   // UNICODE_TO_GBK[9822] := 16#5E62;
   // UNICODE_TO_GBK[9823] := 16#B4B1;
   // UNICODE_TO_GBK[9824] := 16#5E63;
   // UNICODE_TO_GBK[9825] := 16#8EC5;
   // UNICODE_TO_GBK[9826] := 16#5E64;
   // UNICODE_TO_GBK[9827] := 16#8EC6;
   // UNICODE_TO_GBK[9828] := 16#5E65;
   // UNICODE_TO_GBK[9829] := 16#8EC7;
   // UNICODE_TO_GBK[9830] := 16#5E66;
   // UNICODE_TO_GBK[9831] := 16#8EC8;
   // UNICODE_TO_GBK[9832] := 16#5E67;
   // UNICODE_TO_GBK[9833] := 16#8EC9;
   // UNICODE_TO_GBK[9834] := 16#5E68;
   // UNICODE_TO_GBK[9835] := 16#8ECA;
   // UNICODE_TO_GBK[9836] := 16#5E69;
   // UNICODE_TO_GBK[9837] := 16#8ECB;
   // UNICODE_TO_GBK[9838] := 16#5E6A;
   // UNICODE_TO_GBK[9839] := 16#8ECC;
   // UNICODE_TO_GBK[9840] := 16#5E6B;
   // UNICODE_TO_GBK[9841] := 16#8ECD;
   // UNICODE_TO_GBK[9842] := 16#5E6C;
   // UNICODE_TO_GBK[9843] := 16#8ECE;
   // UNICODE_TO_GBK[9844] := 16#5E6D;
   // UNICODE_TO_GBK[9845] := 16#8ECF;
   // UNICODE_TO_GBK[9846] := 16#5E6E;
   // UNICODE_TO_GBK[9847] := 16#8ED0;
   // UNICODE_TO_GBK[9848] := 16#5E6F;
   // UNICODE_TO_GBK[9849] := 16#8ED1;
   // UNICODE_TO_GBK[9850] := 16#5E70;
   // UNICODE_TO_GBK[9851] := 16#8ED2;
   // UNICODE_TO_GBK[9852] := 16#5E71;
   // UNICODE_TO_GBK[9853] := 16#8ED3;
   // UNICODE_TO_GBK[9854] := 16#5E72;
   // UNICODE_TO_GBK[9855] := 16#B8C9;
   // UNICODE_TO_GBK[9856] := 16#5E73;
   // UNICODE_TO_GBK[9857] := 16#C6BD;
   // UNICODE_TO_GBK[9858] := 16#5E74;
   // UNICODE_TO_GBK[9859] := 16#C4EA;
   // UNICODE_TO_GBK[9860] := 16#5E75;
   // UNICODE_TO_GBK[9861] := 16#8ED4;
   // UNICODE_TO_GBK[9862] := 16#5E76;
   // UNICODE_TO_GBK[9863] := 16#B2A2;
   // UNICODE_TO_GBK[9864] := 16#5E77;
   // UNICODE_TO_GBK[9865] := 16#8ED5;
   // UNICODE_TO_GBK[9866] := 16#5E78;
   // UNICODE_TO_GBK[9867] := 16#D0D2;
   // UNICODE_TO_GBK[9868] := 16#5E79;
   // UNICODE_TO_GBK[9869] := 16#8ED6;
   // UNICODE_TO_GBK[9870] := 16#5E7A;
   // UNICODE_TO_GBK[9871] := 16#E7DB;
   // UNICODE_TO_GBK[9872] := 16#5E7B;
   // UNICODE_TO_GBK[9873] := 16#BBC3;
   // UNICODE_TO_GBK[9874] := 16#5E7C;
   // UNICODE_TO_GBK[9875] := 16#D3D7;
   // UNICODE_TO_GBK[9876] := 16#5E7D;
   // UNICODE_TO_GBK[9877] := 16#D3C4;
   // UNICODE_TO_GBK[9878] := 16#5E7E;
   // UNICODE_TO_GBK[9879] := 16#8ED7;
   // UNICODE_TO_GBK[9880] := 16#5E7F;
   // UNICODE_TO_GBK[9881] := 16#B9E3;
   // UNICODE_TO_GBK[9882] := 16#5E80;
   // UNICODE_TO_GBK[9883] := 16#E2CF;
   // UNICODE_TO_GBK[9884] := 16#5E81;
   // UNICODE_TO_GBK[9885] := 16#8ED8;
   // UNICODE_TO_GBK[9886] := 16#5E82;
   // UNICODE_TO_GBK[9887] := 16#8ED9;
   // UNICODE_TO_GBK[9888] := 16#5E83;
   // UNICODE_TO_GBK[9889] := 16#8EDA;
   // UNICODE_TO_GBK[9890] := 16#5E84;
   // UNICODE_TO_GBK[9891] := 16#D7AF;
   // UNICODE_TO_GBK[9892] := 16#5E85;
   // UNICODE_TO_GBK[9893] := 16#8EDB;
   // UNICODE_TO_GBK[9894] := 16#5E86;
   // UNICODE_TO_GBK[9895] := 16#C7EC;
   // UNICODE_TO_GBK[9896] := 16#5E87;
   // UNICODE_TO_GBK[9897] := 16#B1D3;
   // UNICODE_TO_GBK[9898] := 16#5E88;
   // UNICODE_TO_GBK[9899] := 16#8EDC;
   // UNICODE_TO_GBK[9900] := 16#5E89;
   // UNICODE_TO_GBK[9901] := 16#8EDD;
   // UNICODE_TO_GBK[9902] := 16#5E8A;
   // UNICODE_TO_GBK[9903] := 16#B4B2;
   // UNICODE_TO_GBK[9904] := 16#5E8B;
   // UNICODE_TO_GBK[9905] := 16#E2D1;
   // UNICODE_TO_GBK[9906] := 16#5E8C;
   // UNICODE_TO_GBK[9907] := 16#8EDE;
   // UNICODE_TO_GBK[9908] := 16#5E8D;
   // UNICODE_TO_GBK[9909] := 16#8EDF;
   // UNICODE_TO_GBK[9910] := 16#5E8E;
   // UNICODE_TO_GBK[9911] := 16#8EE0;
   // UNICODE_TO_GBK[9912] := 16#5E8F;
   // UNICODE_TO_GBK[9913] := 16#D0F2;
   // UNICODE_TO_GBK[9914] := 16#5E90;
   // UNICODE_TO_GBK[9915] := 16#C2AE;
   // UNICODE_TO_GBK[9916] := 16#5E91;
   // UNICODE_TO_GBK[9917] := 16#E2D0;
   // UNICODE_TO_GBK[9918] := 16#5E92;
   // UNICODE_TO_GBK[9919] := 16#8EE1;
   // UNICODE_TO_GBK[9920] := 16#5E93;
   // UNICODE_TO_GBK[9921] := 16#BFE2;
   // UNICODE_TO_GBK[9922] := 16#5E94;
   // UNICODE_TO_GBK[9923] := 16#D3A6;
   // UNICODE_TO_GBK[9924] := 16#5E95;
   // UNICODE_TO_GBK[9925] := 16#B5D7;
   // UNICODE_TO_GBK[9926] := 16#5E96;
   // UNICODE_TO_GBK[9927] := 16#E2D2;
   // UNICODE_TO_GBK[9928] := 16#5E97;
   // UNICODE_TO_GBK[9929] := 16#B5EA;
   // UNICODE_TO_GBK[9930] := 16#5E98;
   // UNICODE_TO_GBK[9931] := 16#8EE2;
   // UNICODE_TO_GBK[9932] := 16#5E99;
   // UNICODE_TO_GBK[9933] := 16#C3ED;
   // UNICODE_TO_GBK[9934] := 16#5E9A;
   // UNICODE_TO_GBK[9935] := 16#B8FD;
   // UNICODE_TO_GBK[9936] := 16#5E9B;
   // UNICODE_TO_GBK[9937] := 16#8EE3;
   // UNICODE_TO_GBK[9938] := 16#5E9C;
   // UNICODE_TO_GBK[9939] := 16#B8AE;
   // UNICODE_TO_GBK[9940] := 16#5E9D;
   // UNICODE_TO_GBK[9941] := 16#8EE4;
   // UNICODE_TO_GBK[9942] := 16#5E9E;
   // UNICODE_TO_GBK[9943] := 16#C5D3;
   // UNICODE_TO_GBK[9944] := 16#5E9F;
   // UNICODE_TO_GBK[9945] := 16#B7CF;
   // UNICODE_TO_GBK[9946] := 16#5EA0;
   // UNICODE_TO_GBK[9947] := 16#E2D4;
   // UNICODE_TO_GBK[9948] := 16#5EA1;
   // UNICODE_TO_GBK[9949] := 16#8EE5;
   // UNICODE_TO_GBK[9950] := 16#5EA2;
   // UNICODE_TO_GBK[9951] := 16#8EE6;
   // UNICODE_TO_GBK[9952] := 16#5EA3;
   // UNICODE_TO_GBK[9953] := 16#8EE7;
   // UNICODE_TO_GBK[9954] := 16#5EA4;
   // UNICODE_TO_GBK[9955] := 16#8EE8;
   // UNICODE_TO_GBK[9956] := 16#5EA5;
   // UNICODE_TO_GBK[9957] := 16#E2D3;
   // UNICODE_TO_GBK[9958] := 16#5EA6;
   // UNICODE_TO_GBK[9959] := 16#B6C8;
   // UNICODE_TO_GBK[9960] := 16#5EA7;
   // UNICODE_TO_GBK[9961] := 16#D7F9;
   // UNICODE_TO_GBK[9962] := 16#5EA8;
   // UNICODE_TO_GBK[9963] := 16#8EE9;
   // UNICODE_TO_GBK[9964] := 16#5EA9;
   // UNICODE_TO_GBK[9965] := 16#8EEA;
   // UNICODE_TO_GBK[9966] := 16#5EAA;
   // UNICODE_TO_GBK[9967] := 16#8EEB;
   // UNICODE_TO_GBK[9968] := 16#5EAB;
   // UNICODE_TO_GBK[9969] := 16#8EEC;
   // UNICODE_TO_GBK[9970] := 16#5EAC;
   // UNICODE_TO_GBK[9971] := 16#8EED;
   // UNICODE_TO_GBK[9972] := 16#5EAD;
   // UNICODE_TO_GBK[9973] := 16#CDA5;
   // UNICODE_TO_GBK[9974] := 16#5EAE;
   // UNICODE_TO_GBK[9975] := 16#8EEE;
   // UNICODE_TO_GBK[9976] := 16#5EAF;
   // UNICODE_TO_GBK[9977] := 16#8EEF;
   // UNICODE_TO_GBK[9978] := 16#5EB0;
   // UNICODE_TO_GBK[9979] := 16#8EF0;
   // UNICODE_TO_GBK[9980] := 16#5EB1;
   // UNICODE_TO_GBK[9981] := 16#8EF1;
   // UNICODE_TO_GBK[9982] := 16#5EB2;
   // UNICODE_TO_GBK[9983] := 16#8EF2;
   // UNICODE_TO_GBK[9984] := 16#5EB3;
   // UNICODE_TO_GBK[9985] := 16#E2D8;
   // UNICODE_TO_GBK[9986] := 16#5EB4;
   // UNICODE_TO_GBK[9987] := 16#8EF3;
   // UNICODE_TO_GBK[9988] := 16#5EB5;
   // UNICODE_TO_GBK[9989] := 16#E2D6;
   // UNICODE_TO_GBK[9990] := 16#5EB6;
   // UNICODE_TO_GBK[9991] := 16#CAFC;
   // UNICODE_TO_GBK[9992] := 16#5EB7;
   // UNICODE_TO_GBK[9993] := 16#BFB5;
   // UNICODE_TO_GBK[9994] := 16#5EB8;
   // UNICODE_TO_GBK[9995] := 16#D3B9;
   // UNICODE_TO_GBK[9996] := 16#5EB9;
   // UNICODE_TO_GBK[9997] := 16#E2D5;
   // UNICODE_TO_GBK[9998] := 16#5EBA;
   // UNICODE_TO_GBK[9999] := 16#8EF4;
   // UNICODE_TO_GBK[10000] := 16#5EBB;
   // UNICODE_TO_GBK[10001] := 16#8EF5;
   // UNICODE_TO_GBK[10002] := 16#5EBC;
   // UNICODE_TO_GBK[10003] := 16#8EF6;
   // UNICODE_TO_GBK[10004] := 16#5EBD;
   // UNICODE_TO_GBK[10005] := 16#8EF7;
   // UNICODE_TO_GBK[10006] := 16#5EBE;
   // UNICODE_TO_GBK[10007] := 16#E2D7;
   // UNICODE_TO_GBK[10008] := 16#5EBF;
   // UNICODE_TO_GBK[10009] := 16#8EF8;
   // UNICODE_TO_GBK[10010] := 16#5EC0;
   // UNICODE_TO_GBK[10011] := 16#8EF9;
   // UNICODE_TO_GBK[10012] := 16#5EC1;
   // UNICODE_TO_GBK[10013] := 16#8EFA;
   // UNICODE_TO_GBK[10014] := 16#5EC2;
   // UNICODE_TO_GBK[10015] := 16#8EFB;
   // UNICODE_TO_GBK[10016] := 16#5EC3;
   // UNICODE_TO_GBK[10017] := 16#8EFC;
   // UNICODE_TO_GBK[10018] := 16#5EC4;
   // UNICODE_TO_GBK[10019] := 16#8EFD;
   // UNICODE_TO_GBK[10020] := 16#5EC5;
   // UNICODE_TO_GBK[10021] := 16#8EFE;
   // UNICODE_TO_GBK[10022] := 16#5EC6;
   // UNICODE_TO_GBK[10023] := 16#8F40;
   // UNICODE_TO_GBK[10024] := 16#5EC7;
   // UNICODE_TO_GBK[10025] := 16#8F41;
   // UNICODE_TO_GBK[10026] := 16#5EC8;
   // UNICODE_TO_GBK[10027] := 16#8F42;
   // UNICODE_TO_GBK[10028] := 16#5EC9;
   // UNICODE_TO_GBK[10029] := 16#C1AE;
   // UNICODE_TO_GBK[10030] := 16#5ECA;
   // UNICODE_TO_GBK[10031] := 16#C0C8;
   // UNICODE_TO_GBK[10032] := 16#5ECB;
   // UNICODE_TO_GBK[10033] := 16#8F43;
   // UNICODE_TO_GBK[10034] := 16#5ECC;
   // UNICODE_TO_GBK[10035] := 16#8F44;
   // UNICODE_TO_GBK[10036] := 16#5ECD;
   // UNICODE_TO_GBK[10037] := 16#8F45;
   // UNICODE_TO_GBK[10038] := 16#5ECE;
   // UNICODE_TO_GBK[10039] := 16#8F46;
   // UNICODE_TO_GBK[10040] := 16#5ECF;
   // UNICODE_TO_GBK[10041] := 16#8F47;
   // UNICODE_TO_GBK[10042] := 16#5ED0;
   // UNICODE_TO_GBK[10043] := 16#8F48;
   // UNICODE_TO_GBK[10044] := 16#5ED1;
   // UNICODE_TO_GBK[10045] := 16#E2DB;
   // UNICODE_TO_GBK[10046] := 16#5ED2;
   // UNICODE_TO_GBK[10047] := 16#E2DA;
   // UNICODE_TO_GBK[10048] := 16#5ED3;
   // UNICODE_TO_GBK[10049] := 16#C0AA;
   // UNICODE_TO_GBK[10050] := 16#5ED4;
   // UNICODE_TO_GBK[10051] := 16#8F49;
   // UNICODE_TO_GBK[10052] := 16#5ED5;
   // UNICODE_TO_GBK[10053] := 16#8F4A;
   // UNICODE_TO_GBK[10054] := 16#5ED6;
   // UNICODE_TO_GBK[10055] := 16#C1CE;
   // UNICODE_TO_GBK[10056] := 16#5ED7;
   // UNICODE_TO_GBK[10057] := 16#8F4B;
   // UNICODE_TO_GBK[10058] := 16#5ED8;
   // UNICODE_TO_GBK[10059] := 16#8F4C;
   // UNICODE_TO_GBK[10060] := 16#5ED9;
   // UNICODE_TO_GBK[10061] := 16#8F4D;
   // UNICODE_TO_GBK[10062] := 16#5EDA;
   // UNICODE_TO_GBK[10063] := 16#8F4E;
   // UNICODE_TO_GBK[10064] := 16#5EDB;
   // UNICODE_TO_GBK[10065] := 16#E2DC;
   // UNICODE_TO_GBK[10066] := 16#5EDC;
   // UNICODE_TO_GBK[10067] := 16#8F4F;
   // UNICODE_TO_GBK[10068] := 16#5EDD;
   // UNICODE_TO_GBK[10069] := 16#8F50;
   // UNICODE_TO_GBK[10070] := 16#5EDE;
   // UNICODE_TO_GBK[10071] := 16#8F51;
   // UNICODE_TO_GBK[10072] := 16#5EDF;
   // UNICODE_TO_GBK[10073] := 16#8F52;
   // UNICODE_TO_GBK[10074] := 16#5EE0;
   // UNICODE_TO_GBK[10075] := 16#8F53;
   // UNICODE_TO_GBK[10076] := 16#5EE1;
   // UNICODE_TO_GBK[10077] := 16#8F54;
   // UNICODE_TO_GBK[10078] := 16#5EE2;
   // UNICODE_TO_GBK[10079] := 16#8F55;
   // UNICODE_TO_GBK[10080] := 16#5EE3;
   // UNICODE_TO_GBK[10081] := 16#8F56;
   // UNICODE_TO_GBK[10082] := 16#5EE4;
   // UNICODE_TO_GBK[10083] := 16#8F57;
   // UNICODE_TO_GBK[10084] := 16#5EE5;
   // UNICODE_TO_GBK[10085] := 16#8F58;
   // UNICODE_TO_GBK[10086] := 16#5EE6;
   // UNICODE_TO_GBK[10087] := 16#8F59;
   // UNICODE_TO_GBK[10088] := 16#5EE7;
   // UNICODE_TO_GBK[10089] := 16#8F5A;
   // UNICODE_TO_GBK[10090] := 16#5EE8;
   // UNICODE_TO_GBK[10091] := 16#E2DD;
   // UNICODE_TO_GBK[10092] := 16#5EE9;
   // UNICODE_TO_GBK[10093] := 16#8F5B;
   // UNICODE_TO_GBK[10094] := 16#5EEA;
   // UNICODE_TO_GBK[10095] := 16#E2DE;
   // UNICODE_TO_GBK[10096] := 16#5EEB;
   // UNICODE_TO_GBK[10097] := 16#8F5C;
   // UNICODE_TO_GBK[10098] := 16#5EEC;
   // UNICODE_TO_GBK[10099] := 16#8F5D;
   // UNICODE_TO_GBK[10100] := 16#5EED;
   // UNICODE_TO_GBK[10101] := 16#8F5E;
   // UNICODE_TO_GBK[10102] := 16#5EEE;
   // UNICODE_TO_GBK[10103] := 16#8F5F;
   // UNICODE_TO_GBK[10104] := 16#5EEF;
   // UNICODE_TO_GBK[10105] := 16#8F60;
   // UNICODE_TO_GBK[10106] := 16#5EF0;
   // UNICODE_TO_GBK[10107] := 16#8F61;
   // UNICODE_TO_GBK[10108] := 16#5EF1;
   // UNICODE_TO_GBK[10109] := 16#8F62;
   // UNICODE_TO_GBK[10110] := 16#5EF2;
   // UNICODE_TO_GBK[10111] := 16#8F63;
   // UNICODE_TO_GBK[10112] := 16#5EF3;
   // UNICODE_TO_GBK[10113] := 16#8F64;
   // UNICODE_TO_GBK[10114] := 16#5EF4;
   // UNICODE_TO_GBK[10115] := 16#DBC8;
   // UNICODE_TO_GBK[10116] := 16#5EF5;
   // UNICODE_TO_GBK[10117] := 16#8F65;
   // UNICODE_TO_GBK[10118] := 16#5EF6;
   // UNICODE_TO_GBK[10119] := 16#D1D3;
   // UNICODE_TO_GBK[10120] := 16#5EF7;
   // UNICODE_TO_GBK[10121] := 16#CDA2;
   // UNICODE_TO_GBK[10122] := 16#5EF8;
   // UNICODE_TO_GBK[10123] := 16#8F66;
   // UNICODE_TO_GBK[10124] := 16#5EF9;
   // UNICODE_TO_GBK[10125] := 16#8F67;
   // UNICODE_TO_GBK[10126] := 16#5EFA;
   // UNICODE_TO_GBK[10127] := 16#BDA8;
   // UNICODE_TO_GBK[10128] := 16#5EFB;
   // UNICODE_TO_GBK[10129] := 16#8F68;
   // UNICODE_TO_GBK[10130] := 16#5EFC;
   // UNICODE_TO_GBK[10131] := 16#8F69;
   // UNICODE_TO_GBK[10132] := 16#5EFD;
   // UNICODE_TO_GBK[10133] := 16#8F6A;
   // UNICODE_TO_GBK[10134] := 16#5EFE;
   // UNICODE_TO_GBK[10135] := 16#DEC3;
   // UNICODE_TO_GBK[10136] := 16#5EFF;
   // UNICODE_TO_GBK[10137] := 16#D8A5;
   // UNICODE_TO_GBK[10138] := 16#5F00;
   // UNICODE_TO_GBK[10139] := 16#BFAA;
   // UNICODE_TO_GBK[10140] := 16#5F01;
   // UNICODE_TO_GBK[10141] := 16#DBCD;
   // UNICODE_TO_GBK[10142] := 16#5F02;
   // UNICODE_TO_GBK[10143] := 16#D2EC;
   // UNICODE_TO_GBK[10144] := 16#5F03;
   // UNICODE_TO_GBK[10145] := 16#C6FA;
   // UNICODE_TO_GBK[10146] := 16#5F04;
   // UNICODE_TO_GBK[10147] := 16#C5AA;
   // UNICODE_TO_GBK[10148] := 16#5F05;
   // UNICODE_TO_GBK[10149] := 16#8F6B;
   // UNICODE_TO_GBK[10150] := 16#5F06;
   // UNICODE_TO_GBK[10151] := 16#8F6C;
   // UNICODE_TO_GBK[10152] := 16#5F07;
   // UNICODE_TO_GBK[10153] := 16#8F6D;
   // UNICODE_TO_GBK[10154] := 16#5F08;
   // UNICODE_TO_GBK[10155] := 16#DEC4;
   // UNICODE_TO_GBK[10156] := 16#5F09;
   // UNICODE_TO_GBK[10157] := 16#8F6E;
   // UNICODE_TO_GBK[10158] := 16#5F0A;
   // UNICODE_TO_GBK[10159] := 16#B1D7;
   // UNICODE_TO_GBK[10160] := 16#5F0B;
   // UNICODE_TO_GBK[10161] := 16#DFAE;
   // UNICODE_TO_GBK[10162] := 16#5F0C;
   // UNICODE_TO_GBK[10163] := 16#8F6F;
   // UNICODE_TO_GBK[10164] := 16#5F0D;
   // UNICODE_TO_GBK[10165] := 16#8F70;
   // UNICODE_TO_GBK[10166] := 16#5F0E;
   // UNICODE_TO_GBK[10167] := 16#8F71;
   // UNICODE_TO_GBK[10168] := 16#5F0F;
   // UNICODE_TO_GBK[10169] := 16#CABD;
   // UNICODE_TO_GBK[10170] := 16#5F10;
   // UNICODE_TO_GBK[10171] := 16#8F72;
   // UNICODE_TO_GBK[10172] := 16#5F11;
   // UNICODE_TO_GBK[10173] := 16#DFB1;
   // UNICODE_TO_GBK[10174] := 16#5F12;
   // UNICODE_TO_GBK[10175] := 16#8F73;
   // UNICODE_TO_GBK[10176] := 16#5F13;
   // UNICODE_TO_GBK[10177] := 16#B9AD;
   // UNICODE_TO_GBK[10178] := 16#5F14;
   // UNICODE_TO_GBK[10179] := 16#8F74;
   // UNICODE_TO_GBK[10180] := 16#5F15;
   // UNICODE_TO_GBK[10181] := 16#D2FD;
   // UNICODE_TO_GBK[10182] := 16#5F16;
   // UNICODE_TO_GBK[10183] := 16#8F75;
   // UNICODE_TO_GBK[10184] := 16#5F17;
   // UNICODE_TO_GBK[10185] := 16#B8A5;
   // UNICODE_TO_GBK[10186] := 16#5F18;
   // UNICODE_TO_GBK[10187] := 16#BAEB;
   // UNICODE_TO_GBK[10188] := 16#5F19;
   // UNICODE_TO_GBK[10189] := 16#8F76;
   // UNICODE_TO_GBK[10190] := 16#5F1A;
   // UNICODE_TO_GBK[10191] := 16#8F77;
   // UNICODE_TO_GBK[10192] := 16#5F1B;
   // UNICODE_TO_GBK[10193] := 16#B3DA;
   // UNICODE_TO_GBK[10194] := 16#5F1C;
   // UNICODE_TO_GBK[10195] := 16#8F78;
   // UNICODE_TO_GBK[10196] := 16#5F1D;
   // UNICODE_TO_GBK[10197] := 16#8F79;
   // UNICODE_TO_GBK[10198] := 16#5F1E;
   // UNICODE_TO_GBK[10199] := 16#8F7A;
   // UNICODE_TO_GBK[10200] := 16#5F1F;
   // UNICODE_TO_GBK[10201] := 16#B5DC;
   // UNICODE_TO_GBK[10202] := 16#5F20;
   // UNICODE_TO_GBK[10203] := 16#D5C5;
   // UNICODE_TO_GBK[10204] := 16#5F21;
   // UNICODE_TO_GBK[10205] := 16#8F7B;
   // UNICODE_TO_GBK[10206] := 16#5F22;
   // UNICODE_TO_GBK[10207] := 16#8F7C;
   // UNICODE_TO_GBK[10208] := 16#5F23;
   // UNICODE_TO_GBK[10209] := 16#8F7D;
   // UNICODE_TO_GBK[10210] := 16#5F24;
   // UNICODE_TO_GBK[10211] := 16#8F7E;
   // UNICODE_TO_GBK[10212] := 16#5F25;
   // UNICODE_TO_GBK[10213] := 16#C3D6;
   // UNICODE_TO_GBK[10214] := 16#5F26;
   // UNICODE_TO_GBK[10215] := 16#CFD2;
   // UNICODE_TO_GBK[10216] := 16#5F27;
   // UNICODE_TO_GBK[10217] := 16#BBA1;
   // UNICODE_TO_GBK[10218] := 16#5F28;
   // UNICODE_TO_GBK[10219] := 16#8F80;
   // UNICODE_TO_GBK[10220] := 16#5F29;
   // UNICODE_TO_GBK[10221] := 16#E5F3;
   // UNICODE_TO_GBK[10222] := 16#5F2A;
   // UNICODE_TO_GBK[10223] := 16#E5F2;
   // UNICODE_TO_GBK[10224] := 16#5F2B;
   // UNICODE_TO_GBK[10225] := 16#8F81;
   // UNICODE_TO_GBK[10226] := 16#5F2C;
   // UNICODE_TO_GBK[10227] := 16#8F82;
   // UNICODE_TO_GBK[10228] := 16#5F2D;
   // UNICODE_TO_GBK[10229] := 16#E5F4;
   // UNICODE_TO_GBK[10230] := 16#5F2E;
   // UNICODE_TO_GBK[10231] := 16#8F83;
   // UNICODE_TO_GBK[10232] := 16#5F2F;
   // UNICODE_TO_GBK[10233] := 16#CDE4;
   // UNICODE_TO_GBK[10234] := 16#5F30;
   // UNICODE_TO_GBK[10235] := 16#8F84;
   // UNICODE_TO_GBK[10236] := 16#5F31;
   // UNICODE_TO_GBK[10237] := 16#C8F5;
   // UNICODE_TO_GBK[10238] := 16#5F32;
   // UNICODE_TO_GBK[10239] := 16#8F85;
   // UNICODE_TO_GBK[10240] := 16#5F33;
   // UNICODE_TO_GBK[10241] := 16#8F86;
   // UNICODE_TO_GBK[10242] := 16#5F34;
   // UNICODE_TO_GBK[10243] := 16#8F87;
   // UNICODE_TO_GBK[10244] := 16#5F35;
   // UNICODE_TO_GBK[10245] := 16#8F88;
   // UNICODE_TO_GBK[10246] := 16#5F36;
   // UNICODE_TO_GBK[10247] := 16#8F89;
   // UNICODE_TO_GBK[10248] := 16#5F37;
   // UNICODE_TO_GBK[10249] := 16#8F8A;
   // UNICODE_TO_GBK[10250] := 16#5F38;
   // UNICODE_TO_GBK[10251] := 16#8F8B;
   // UNICODE_TO_GBK[10252] := 16#5F39;
   // UNICODE_TO_GBK[10253] := 16#B5AF;
   // UNICODE_TO_GBK[10254] := 16#5F3A;
   // UNICODE_TO_GBK[10255] := 16#C7BF;
   // UNICODE_TO_GBK[10256] := 16#5F3B;
   // UNICODE_TO_GBK[10257] := 16#8F8C;
   // UNICODE_TO_GBK[10258] := 16#5F3C;
   // UNICODE_TO_GBK[10259] := 16#E5F6;
   // UNICODE_TO_GBK[10260] := 16#5F3D;
   // UNICODE_TO_GBK[10261] := 16#8F8D;
   // UNICODE_TO_GBK[10262] := 16#5F3E;
   // UNICODE_TO_GBK[10263] := 16#8F8E;
   // UNICODE_TO_GBK[10264] := 16#5F3F;
   // UNICODE_TO_GBK[10265] := 16#8F8F;
   // UNICODE_TO_GBK[10266] := 16#5F40;
   // UNICODE_TO_GBK[10267] := 16#ECB0;
   // UNICODE_TO_GBK[10268] := 16#5F41;
   // UNICODE_TO_GBK[10269] := 16#8F90;
   // UNICODE_TO_GBK[10270] := 16#5F42;
   // UNICODE_TO_GBK[10271] := 16#8F91;
   // UNICODE_TO_GBK[10272] := 16#5F43;
   // UNICODE_TO_GBK[10273] := 16#8F92;
   // UNICODE_TO_GBK[10274] := 16#5F44;
   // UNICODE_TO_GBK[10275] := 16#8F93;
   // UNICODE_TO_GBK[10276] := 16#5F45;
   // UNICODE_TO_GBK[10277] := 16#8F94;
   // UNICODE_TO_GBK[10278] := 16#5F46;
   // UNICODE_TO_GBK[10279] := 16#8F95;
   // UNICODE_TO_GBK[10280] := 16#5F47;
   // UNICODE_TO_GBK[10281] := 16#8F96;
   // UNICODE_TO_GBK[10282] := 16#5F48;
   // UNICODE_TO_GBK[10283] := 16#8F97;
   // UNICODE_TO_GBK[10284] := 16#5F49;
   // UNICODE_TO_GBK[10285] := 16#8F98;
   // UNICODE_TO_GBK[10286] := 16#5F4A;
   // UNICODE_TO_GBK[10287] := 16#8F99;
   // UNICODE_TO_GBK[10288] := 16#5F4B;
   // UNICODE_TO_GBK[10289] := 16#8F9A;
   // UNICODE_TO_GBK[10290] := 16#5F4C;
   // UNICODE_TO_GBK[10291] := 16#8F9B;
   // UNICODE_TO_GBK[10292] := 16#5F4D;
   // UNICODE_TO_GBK[10293] := 16#8F9C;
   // UNICODE_TO_GBK[10294] := 16#5F4E;
   // UNICODE_TO_GBK[10295] := 16#8F9D;
   // UNICODE_TO_GBK[10296] := 16#5F4F;
   // UNICODE_TO_GBK[10297] := 16#8F9E;
   // UNICODE_TO_GBK[10298] := 16#5F50;
   // UNICODE_TO_GBK[10299] := 16#E5E6;
   // UNICODE_TO_GBK[10300] := 16#5F51;
   // UNICODE_TO_GBK[10301] := 16#8F9F;
   // UNICODE_TO_GBK[10302] := 16#5F52;
   // UNICODE_TO_GBK[10303] := 16#B9E9;
   // UNICODE_TO_GBK[10304] := 16#5F53;
   // UNICODE_TO_GBK[10305] := 16#B5B1;
   // UNICODE_TO_GBK[10306] := 16#5F54;
   // UNICODE_TO_GBK[10307] := 16#8FA0;
   // UNICODE_TO_GBK[10308] := 16#5F55;
   // UNICODE_TO_GBK[10309] := 16#C2BC;
   // UNICODE_TO_GBK[10310] := 16#5F56;
   // UNICODE_TO_GBK[10311] := 16#E5E8;
   // UNICODE_TO_GBK[10312] := 16#5F57;
   // UNICODE_TO_GBK[10313] := 16#E5E7;
   // UNICODE_TO_GBK[10314] := 16#5F58;
   // UNICODE_TO_GBK[10315] := 16#E5E9;
   // UNICODE_TO_GBK[10316] := 16#5F59;
   // UNICODE_TO_GBK[10317] := 16#8FA1;
   // UNICODE_TO_GBK[10318] := 16#5F5A;
   // UNICODE_TO_GBK[10319] := 16#8FA2;
   // UNICODE_TO_GBK[10320] := 16#5F5B;
   // UNICODE_TO_GBK[10321] := 16#8FA3;
   // UNICODE_TO_GBK[10322] := 16#5F5C;
   // UNICODE_TO_GBK[10323] := 16#8FA4;
   // UNICODE_TO_GBK[10324] := 16#5F5D;
   // UNICODE_TO_GBK[10325] := 16#D2CD;
   // UNICODE_TO_GBK[10326] := 16#5F5E;
   // UNICODE_TO_GBK[10327] := 16#8FA5;
   // UNICODE_TO_GBK[10328] := 16#5F5F;
   // UNICODE_TO_GBK[10329] := 16#8FA6;
   // UNICODE_TO_GBK[10330] := 16#5F60;
   // UNICODE_TO_GBK[10331] := 16#8FA7;
   // UNICODE_TO_GBK[10332] := 16#5F61;
   // UNICODE_TO_GBK[10333] := 16#E1EA;
   // UNICODE_TO_GBK[10334] := 16#5F62;
   // UNICODE_TO_GBK[10335] := 16#D0CE;
   // UNICODE_TO_GBK[10336] := 16#5F63;
   // UNICODE_TO_GBK[10337] := 16#8FA8;
   // UNICODE_TO_GBK[10338] := 16#5F64;
   // UNICODE_TO_GBK[10339] := 16#CDAE;
   // UNICODE_TO_GBK[10340] := 16#5F65;
   // UNICODE_TO_GBK[10341] := 16#8FA9;
   // UNICODE_TO_GBK[10342] := 16#5F66;
   // UNICODE_TO_GBK[10343] := 16#D1E5;
   // UNICODE_TO_GBK[10344] := 16#5F67;
   // UNICODE_TO_GBK[10345] := 16#8FAA;
   // UNICODE_TO_GBK[10346] := 16#5F68;
   // UNICODE_TO_GBK[10347] := 16#8FAB;
   // UNICODE_TO_GBK[10348] := 16#5F69;
   // UNICODE_TO_GBK[10349] := 16#B2CA;
   // UNICODE_TO_GBK[10350] := 16#5F6A;
   // UNICODE_TO_GBK[10351] := 16#B1EB;
   // UNICODE_TO_GBK[10352] := 16#5F6B;
   // UNICODE_TO_GBK[10353] := 16#8FAC;
   // UNICODE_TO_GBK[10354] := 16#5F6C;
   // UNICODE_TO_GBK[10355] := 16#B1F2;
   // UNICODE_TO_GBK[10356] := 16#5F6D;
   // UNICODE_TO_GBK[10357] := 16#C5ED;
   // UNICODE_TO_GBK[10358] := 16#5F6E;
   // UNICODE_TO_GBK[10359] := 16#8FAD;
   // UNICODE_TO_GBK[10360] := 16#5F6F;
   // UNICODE_TO_GBK[10361] := 16#8FAE;
   // UNICODE_TO_GBK[10362] := 16#5F70;
   // UNICODE_TO_GBK[10363] := 16#D5C3;
   // UNICODE_TO_GBK[10364] := 16#5F71;
   // UNICODE_TO_GBK[10365] := 16#D3B0;
   // UNICODE_TO_GBK[10366] := 16#5F72;
   // UNICODE_TO_GBK[10367] := 16#8FAF;
   // UNICODE_TO_GBK[10368] := 16#5F73;
   // UNICODE_TO_GBK[10369] := 16#E1DC;
   // UNICODE_TO_GBK[10370] := 16#5F74;
   // UNICODE_TO_GBK[10371] := 16#8FB0;
   // UNICODE_TO_GBK[10372] := 16#5F75;
   // UNICODE_TO_GBK[10373] := 16#8FB1;
   // UNICODE_TO_GBK[10374] := 16#5F76;
   // UNICODE_TO_GBK[10375] := 16#8FB2;
   // UNICODE_TO_GBK[10376] := 16#5F77;
   // UNICODE_TO_GBK[10377] := 16#E1DD;
   // UNICODE_TO_GBK[10378] := 16#5F78;
   // UNICODE_TO_GBK[10379] := 16#8FB3;
   // UNICODE_TO_GBK[10380] := 16#5F79;
   // UNICODE_TO_GBK[10381] := 16#D2DB;
   // UNICODE_TO_GBK[10382] := 16#5F7A;
   // UNICODE_TO_GBK[10383] := 16#8FB4;
   // UNICODE_TO_GBK[10384] := 16#5F7B;
   // UNICODE_TO_GBK[10385] := 16#B3B9;
   // UNICODE_TO_GBK[10386] := 16#5F7C;
   // UNICODE_TO_GBK[10387] := 16#B1CB;
   // UNICODE_TO_GBK[10388] := 16#5F7D;
   // UNICODE_TO_GBK[10389] := 16#8FB5;
   // UNICODE_TO_GBK[10390] := 16#5F7E;
   // UNICODE_TO_GBK[10391] := 16#8FB6;
   // UNICODE_TO_GBK[10392] := 16#5F7F;
   // UNICODE_TO_GBK[10393] := 16#8FB7;
   // UNICODE_TO_GBK[10394] := 16#5F80;
   // UNICODE_TO_GBK[10395] := 16#CDF9;
   // UNICODE_TO_GBK[10396] := 16#5F81;
   // UNICODE_TO_GBK[10397] := 16#D5F7;
   // UNICODE_TO_GBK[10398] := 16#5F82;
   // UNICODE_TO_GBK[10399] := 16#E1DE;
   // UNICODE_TO_GBK[10400] := 16#5F83;
   // UNICODE_TO_GBK[10401] := 16#8FB8;
   // UNICODE_TO_GBK[10402] := 16#5F84;
   // UNICODE_TO_GBK[10403] := 16#BEB6;
   // UNICODE_TO_GBK[10404] := 16#5F85;
   // UNICODE_TO_GBK[10405] := 16#B4FD;
   // UNICODE_TO_GBK[10406] := 16#5F86;
   // UNICODE_TO_GBK[10407] := 16#8FB9;
   // UNICODE_TO_GBK[10408] := 16#5F87;
   // UNICODE_TO_GBK[10409] := 16#E1DF;
   // UNICODE_TO_GBK[10410] := 16#5F88;
   // UNICODE_TO_GBK[10411] := 16#BADC;
   // UNICODE_TO_GBK[10412] := 16#5F89;
   // UNICODE_TO_GBK[10413] := 16#E1E0;
   // UNICODE_TO_GBK[10414] := 16#5F8A;
   // UNICODE_TO_GBK[10415] := 16#BBB2;
   // UNICODE_TO_GBK[10416] := 16#5F8B;
   // UNICODE_TO_GBK[10417] := 16#C2C9;
   // UNICODE_TO_GBK[10418] := 16#5F8C;
   // UNICODE_TO_GBK[10419] := 16#E1E1;
   // UNICODE_TO_GBK[10420] := 16#5F8D;
   // UNICODE_TO_GBK[10421] := 16#8FBA;
   // UNICODE_TO_GBK[10422] := 16#5F8E;
   // UNICODE_TO_GBK[10423] := 16#8FBB;
   // UNICODE_TO_GBK[10424] := 16#5F8F;
   // UNICODE_TO_GBK[10425] := 16#8FBC;
   // UNICODE_TO_GBK[10426] := 16#5F90;
   // UNICODE_TO_GBK[10427] := 16#D0EC;
   // UNICODE_TO_GBK[10428] := 16#5F91;
   // UNICODE_TO_GBK[10429] := 16#8FBD;
   // UNICODE_TO_GBK[10430] := 16#5F92;
   // UNICODE_TO_GBK[10431] := 16#CDBD;
   // UNICODE_TO_GBK[10432] := 16#5F93;
   // UNICODE_TO_GBK[10433] := 16#8FBE;
   // UNICODE_TO_GBK[10434] := 16#5F94;
   // UNICODE_TO_GBK[10435] := 16#8FBF;
   // UNICODE_TO_GBK[10436] := 16#5F95;
   // UNICODE_TO_GBK[10437] := 16#E1E2;
   // UNICODE_TO_GBK[10438] := 16#5F96;
   // UNICODE_TO_GBK[10439] := 16#8FC0;
   // UNICODE_TO_GBK[10440] := 16#5F97;
   // UNICODE_TO_GBK[10441] := 16#B5C3;
   // UNICODE_TO_GBK[10442] := 16#5F98;
   // UNICODE_TO_GBK[10443] := 16#C5C7;
   // UNICODE_TO_GBK[10444] := 16#5F99;
   // UNICODE_TO_GBK[10445] := 16#E1E3;
   // UNICODE_TO_GBK[10446] := 16#5F9A;
   // UNICODE_TO_GBK[10447] := 16#8FC1;
   // UNICODE_TO_GBK[10448] := 16#5F9B;
   // UNICODE_TO_GBK[10449] := 16#8FC2;
   // UNICODE_TO_GBK[10450] := 16#5F9C;
   // UNICODE_TO_GBK[10451] := 16#E1E4;
   // UNICODE_TO_GBK[10452] := 16#5F9D;
   // UNICODE_TO_GBK[10453] := 16#8FC3;
   // UNICODE_TO_GBK[10454] := 16#5F9E;
   // UNICODE_TO_GBK[10455] := 16#8FC4;
   // UNICODE_TO_GBK[10456] := 16#5F9F;
   // UNICODE_TO_GBK[10457] := 16#8FC5;
   // UNICODE_TO_GBK[10458] := 16#5FA0;
   // UNICODE_TO_GBK[10459] := 16#8FC6;
   // UNICODE_TO_GBK[10460] := 16#5FA1;
   // UNICODE_TO_GBK[10461] := 16#D3F9;
   // UNICODE_TO_GBK[10462] := 16#5FA2;
   // UNICODE_TO_GBK[10463] := 16#8FC7;
   // UNICODE_TO_GBK[10464] := 16#5FA3;
   // UNICODE_TO_GBK[10465] := 16#8FC8;
   // UNICODE_TO_GBK[10466] := 16#5FA4;
   // UNICODE_TO_GBK[10467] := 16#8FC9;
   // UNICODE_TO_GBK[10468] := 16#5FA5;
   // UNICODE_TO_GBK[10469] := 16#8FCA;
   // UNICODE_TO_GBK[10470] := 16#5FA6;
   // UNICODE_TO_GBK[10471] := 16#8FCB;
   // UNICODE_TO_GBK[10472] := 16#5FA7;
   // UNICODE_TO_GBK[10473] := 16#8FCC;
   // UNICODE_TO_GBK[10474] := 16#5FA8;
   // UNICODE_TO_GBK[10475] := 16#E1E5;
   // UNICODE_TO_GBK[10476] := 16#5FA9;
   // UNICODE_TO_GBK[10477] := 16#8FCD;
   // UNICODE_TO_GBK[10478] := 16#5FAA;
   // UNICODE_TO_GBK[10479] := 16#D1AD;
   // UNICODE_TO_GBK[10480] := 16#5FAB;
   // UNICODE_TO_GBK[10481] := 16#8FCE;
   // UNICODE_TO_GBK[10482] := 16#5FAC;
   // UNICODE_TO_GBK[10483] := 16#8FCF;
   // UNICODE_TO_GBK[10484] := 16#5FAD;
   // UNICODE_TO_GBK[10485] := 16#E1E6;
   // UNICODE_TO_GBK[10486] := 16#5FAE;
   // UNICODE_TO_GBK[10487] := 16#CEA2;
   // UNICODE_TO_GBK[10488] := 16#5FAF;
   // UNICODE_TO_GBK[10489] := 16#8FD0;
   // UNICODE_TO_GBK[10490] := 16#5FB0;
   // UNICODE_TO_GBK[10491] := 16#8FD1;
   // UNICODE_TO_GBK[10492] := 16#5FB1;
   // UNICODE_TO_GBK[10493] := 16#8FD2;
   // UNICODE_TO_GBK[10494] := 16#5FB2;
   // UNICODE_TO_GBK[10495] := 16#8FD3;
   // UNICODE_TO_GBK[10496] := 16#5FB3;
   // UNICODE_TO_GBK[10497] := 16#8FD4;
   // UNICODE_TO_GBK[10498] := 16#5FB4;
   // UNICODE_TO_GBK[10499] := 16#8FD5;
   // UNICODE_TO_GBK[10500] := 16#5FB5;
   // UNICODE_TO_GBK[10501] := 16#E1E7;
   // UNICODE_TO_GBK[10502] := 16#5FB6;
   // UNICODE_TO_GBK[10503] := 16#8FD6;
   // UNICODE_TO_GBK[10504] := 16#5FB7;
   // UNICODE_TO_GBK[10505] := 16#B5C2;
   // UNICODE_TO_GBK[10506] := 16#5FB8;
   // UNICODE_TO_GBK[10507] := 16#8FD7;
   // UNICODE_TO_GBK[10508] := 16#5FB9;
   // UNICODE_TO_GBK[10509] := 16#8FD8;
   // UNICODE_TO_GBK[10510] := 16#5FBA;
   // UNICODE_TO_GBK[10511] := 16#8FD9;
   // UNICODE_TO_GBK[10512] := 16#5FBB;
   // UNICODE_TO_GBK[10513] := 16#8FDA;
   // UNICODE_TO_GBK[10514] := 16#5FBC;
   // UNICODE_TO_GBK[10515] := 16#E1E8;
   // UNICODE_TO_GBK[10516] := 16#5FBD;
   // UNICODE_TO_GBK[10517] := 16#BBD5;
   // UNICODE_TO_GBK[10518] := 16#5FBE;
   // UNICODE_TO_GBK[10519] := 16#8FDB;
   // UNICODE_TO_GBK[10520] := 16#5FBF;
   // UNICODE_TO_GBK[10521] := 16#8FDC;
   // UNICODE_TO_GBK[10522] := 16#5FC0;
   // UNICODE_TO_GBK[10523] := 16#8FDD;
   // UNICODE_TO_GBK[10524] := 16#5FC1;
   // UNICODE_TO_GBK[10525] := 16#8FDE;
   // UNICODE_TO_GBK[10526] := 16#5FC2;
   // UNICODE_TO_GBK[10527] := 16#8FDF;
   // UNICODE_TO_GBK[10528] := 16#5FC3;
   // UNICODE_TO_GBK[10529] := 16#D0C4;
   // UNICODE_TO_GBK[10530] := 16#5FC4;
   // UNICODE_TO_GBK[10531] := 16#E2E0;
   // UNICODE_TO_GBK[10532] := 16#5FC5;
   // UNICODE_TO_GBK[10533] := 16#B1D8;
   // UNICODE_TO_GBK[10534] := 16#5FC6;
   // UNICODE_TO_GBK[10535] := 16#D2E4;
   // UNICODE_TO_GBK[10536] := 16#5FC7;
   // UNICODE_TO_GBK[10537] := 16#8FE0;
   // UNICODE_TO_GBK[10538] := 16#5FC8;
   // UNICODE_TO_GBK[10539] := 16#8FE1;
   // UNICODE_TO_GBK[10540] := 16#5FC9;
   // UNICODE_TO_GBK[10541] := 16#E2E1;
   // UNICODE_TO_GBK[10542] := 16#5FCA;
   // UNICODE_TO_GBK[10543] := 16#8FE2;
   // UNICODE_TO_GBK[10544] := 16#5FCB;
   // UNICODE_TO_GBK[10545] := 16#8FE3;
   // UNICODE_TO_GBK[10546] := 16#5FCC;
   // UNICODE_TO_GBK[10547] := 16#BCC9;
   // UNICODE_TO_GBK[10548] := 16#5FCD;
   // UNICODE_TO_GBK[10549] := 16#C8CC;
   // UNICODE_TO_GBK[10550] := 16#5FCE;
   // UNICODE_TO_GBK[10551] := 16#8FE4;
   // UNICODE_TO_GBK[10552] := 16#5FCF;
   // UNICODE_TO_GBK[10553] := 16#E2E3;
   // UNICODE_TO_GBK[10554] := 16#5FD0;
   // UNICODE_TO_GBK[10555] := 16#ECFE;
   // UNICODE_TO_GBK[10556] := 16#5FD1;
   // UNICODE_TO_GBK[10557] := 16#ECFD;
   // UNICODE_TO_GBK[10558] := 16#5FD2;
   // UNICODE_TO_GBK[10559] := 16#DFAF;
   // UNICODE_TO_GBK[10560] := 16#5FD3;
   // UNICODE_TO_GBK[10561] := 16#8FE5;
   // UNICODE_TO_GBK[10562] := 16#5FD4;
   // UNICODE_TO_GBK[10563] := 16#8FE6;
   // UNICODE_TO_GBK[10564] := 16#5FD5;
   // UNICODE_TO_GBK[10565] := 16#8FE7;
   // UNICODE_TO_GBK[10566] := 16#5FD6;
   // UNICODE_TO_GBK[10567] := 16#E2E2;
   // UNICODE_TO_GBK[10568] := 16#5FD7;
   // UNICODE_TO_GBK[10569] := 16#D6BE;
   // UNICODE_TO_GBK[10570] := 16#5FD8;
   // UNICODE_TO_GBK[10571] := 16#CDFC;
   // UNICODE_TO_GBK[10572] := 16#5FD9;
   // UNICODE_TO_GBK[10573] := 16#C3A6;
   // UNICODE_TO_GBK[10574] := 16#5FDA;
   // UNICODE_TO_GBK[10575] := 16#8FE8;
   // UNICODE_TO_GBK[10576] := 16#5FDB;
   // UNICODE_TO_GBK[10577] := 16#8FE9;
   // UNICODE_TO_GBK[10578] := 16#5FDC;
   // UNICODE_TO_GBK[10579] := 16#8FEA;
   // UNICODE_TO_GBK[10580] := 16#5FDD;
   // UNICODE_TO_GBK[10581] := 16#E3C3;
   // UNICODE_TO_GBK[10582] := 16#5FDE;
   // UNICODE_TO_GBK[10583] := 16#8FEB;
   // UNICODE_TO_GBK[10584] := 16#5FDF;
   // UNICODE_TO_GBK[10585] := 16#8FEC;
   // UNICODE_TO_GBK[10586] := 16#5FE0;
   // UNICODE_TO_GBK[10587] := 16#D6D2;
   // UNICODE_TO_GBK[10588] := 16#5FE1;
   // UNICODE_TO_GBK[10589] := 16#E2E7;
   // UNICODE_TO_GBK[10590] := 16#5FE2;
   // UNICODE_TO_GBK[10591] := 16#8FED;
   // UNICODE_TO_GBK[10592] := 16#5FE3;
   // UNICODE_TO_GBK[10593] := 16#8FEE;
   // UNICODE_TO_GBK[10594] := 16#5FE4;
   // UNICODE_TO_GBK[10595] := 16#E2E8;
   // UNICODE_TO_GBK[10596] := 16#5FE5;
   // UNICODE_TO_GBK[10597] := 16#8FEF;
   // UNICODE_TO_GBK[10598] := 16#5FE6;
   // UNICODE_TO_GBK[10599] := 16#8FF0;
   // UNICODE_TO_GBK[10600] := 16#5FE7;
   // UNICODE_TO_GBK[10601] := 16#D3C7;
   // UNICODE_TO_GBK[10602] := 16#5FE8;
   // UNICODE_TO_GBK[10603] := 16#8FF1;
   // UNICODE_TO_GBK[10604] := 16#5FE9;
   // UNICODE_TO_GBK[10605] := 16#8FF2;
   // UNICODE_TO_GBK[10606] := 16#5FEA;
   // UNICODE_TO_GBK[10607] := 16#E2EC;
   // UNICODE_TO_GBK[10608] := 16#5FEB;
   // UNICODE_TO_GBK[10609] := 16#BFEC;
   // UNICODE_TO_GBK[10610] := 16#5FEC;
   // UNICODE_TO_GBK[10611] := 16#8FF3;
   // UNICODE_TO_GBK[10612] := 16#5FED;
   // UNICODE_TO_GBK[10613] := 16#E2ED;
   // UNICODE_TO_GBK[10614] := 16#5FEE;
   // UNICODE_TO_GBK[10615] := 16#E2E5;
   // UNICODE_TO_GBK[10616] := 16#5FEF;
   // UNICODE_TO_GBK[10617] := 16#8FF4;
   // UNICODE_TO_GBK[10618] := 16#5FF0;
   // UNICODE_TO_GBK[10619] := 16#8FF5;
   // UNICODE_TO_GBK[10620] := 16#5FF1;
   // UNICODE_TO_GBK[10621] := 16#B3C0;
   // UNICODE_TO_GBK[10622] := 16#5FF2;
   // UNICODE_TO_GBK[10623] := 16#8FF6;
   // UNICODE_TO_GBK[10624] := 16#5FF3;
   // UNICODE_TO_GBK[10625] := 16#8FF7;
   // UNICODE_TO_GBK[10626] := 16#5FF4;
   // UNICODE_TO_GBK[10627] := 16#8FF8;
   // UNICODE_TO_GBK[10628] := 16#5FF5;
   // UNICODE_TO_GBK[10629] := 16#C4EE;
   // UNICODE_TO_GBK[10630] := 16#5FF6;
   // UNICODE_TO_GBK[10631] := 16#8FF9;
   // UNICODE_TO_GBK[10632] := 16#5FF7;
   // UNICODE_TO_GBK[10633] := 16#8FFA;
   // UNICODE_TO_GBK[10634] := 16#5FF8;
   // UNICODE_TO_GBK[10635] := 16#E2EE;
   // UNICODE_TO_GBK[10636] := 16#5FF9;
   // UNICODE_TO_GBK[10637] := 16#8FFB;
   // UNICODE_TO_GBK[10638] := 16#5FFA;
   // UNICODE_TO_GBK[10639] := 16#8FFC;
   // UNICODE_TO_GBK[10640] := 16#5FFB;
   // UNICODE_TO_GBK[10641] := 16#D0C3;
   // UNICODE_TO_GBK[10642] := 16#5FFC;
   // UNICODE_TO_GBK[10643] := 16#8FFD;
   // UNICODE_TO_GBK[10644] := 16#5FFD;
   // UNICODE_TO_GBK[10645] := 16#BAF6;
   // UNICODE_TO_GBK[10646] := 16#5FFE;
   // UNICODE_TO_GBK[10647] := 16#E2E9;
   // UNICODE_TO_GBK[10648] := 16#5FFF;
   // UNICODE_TO_GBK[10649] := 16#B7DE;
   // UNICODE_TO_GBK[10650] := 16#6000;
   // UNICODE_TO_GBK[10651] := 16#BBB3;
   // UNICODE_TO_GBK[10652] := 16#6001;
   // UNICODE_TO_GBK[10653] := 16#CCAC;
   // UNICODE_TO_GBK[10654] := 16#6002;
   // UNICODE_TO_GBK[10655] := 16#CBCB;
   // UNICODE_TO_GBK[10656] := 16#6003;
   // UNICODE_TO_GBK[10657] := 16#E2E4;
   // UNICODE_TO_GBK[10658] := 16#6004;
   // UNICODE_TO_GBK[10659] := 16#E2E6;
   // UNICODE_TO_GBK[10660] := 16#6005;
   // UNICODE_TO_GBK[10661] := 16#E2EA;
   // UNICODE_TO_GBK[10662] := 16#6006;
   // UNICODE_TO_GBK[10663] := 16#E2EB;
   // UNICODE_TO_GBK[10664] := 16#6007;
   // UNICODE_TO_GBK[10665] := 16#8FFE;
   // UNICODE_TO_GBK[10666] := 16#6008;
   // UNICODE_TO_GBK[10667] := 16#9040;
   // UNICODE_TO_GBK[10668] := 16#6009;
   // UNICODE_TO_GBK[10669] := 16#9041;
   // UNICODE_TO_GBK[10670] := 16#600A;
   // UNICODE_TO_GBK[10671] := 16#E2F7;
   // UNICODE_TO_GBK[10672] := 16#600B;
   // UNICODE_TO_GBK[10673] := 16#9042;
   // UNICODE_TO_GBK[10674] := 16#600C;
   // UNICODE_TO_GBK[10675] := 16#9043;
   // UNICODE_TO_GBK[10676] := 16#600D;
   // UNICODE_TO_GBK[10677] := 16#E2F4;
   // UNICODE_TO_GBK[10678] := 16#600E;
   // UNICODE_TO_GBK[10679] := 16#D4F5;
   // UNICODE_TO_GBK[10680] := 16#600F;
   // UNICODE_TO_GBK[10681] := 16#E2F3;
   // UNICODE_TO_GBK[10682] := 16#6010;
   // UNICODE_TO_GBK[10683] := 16#9044;
   // UNICODE_TO_GBK[10684] := 16#6011;
   // UNICODE_TO_GBK[10685] := 16#9045;
   // UNICODE_TO_GBK[10686] := 16#6012;
   // UNICODE_TO_GBK[10687] := 16#C5AD;
   // UNICODE_TO_GBK[10688] := 16#6013;
   // UNICODE_TO_GBK[10689] := 16#9046;
   // UNICODE_TO_GBK[10690] := 16#6014;
   // UNICODE_TO_GBK[10691] := 16#D5FA;
   // UNICODE_TO_GBK[10692] := 16#6015;
   // UNICODE_TO_GBK[10693] := 16#C5C2;
   // UNICODE_TO_GBK[10694] := 16#6016;
   // UNICODE_TO_GBK[10695] := 16#B2C0;
   // UNICODE_TO_GBK[10696] := 16#6017;
   // UNICODE_TO_GBK[10697] := 16#9047;
   // UNICODE_TO_GBK[10698] := 16#6018;
   // UNICODE_TO_GBK[10699] := 16#9048;
   // UNICODE_TO_GBK[10700] := 16#6019;
   // UNICODE_TO_GBK[10701] := 16#E2EF;
   // UNICODE_TO_GBK[10702] := 16#601A;
   // UNICODE_TO_GBK[10703] := 16#9049;
   // UNICODE_TO_GBK[10704] := 16#601B;
   // UNICODE_TO_GBK[10705] := 16#E2F2;
   // UNICODE_TO_GBK[10706] := 16#601C;
   // UNICODE_TO_GBK[10707] := 16#C1AF;
   // UNICODE_TO_GBK[10708] := 16#601D;
   // UNICODE_TO_GBK[10709] := 16#CBBC;
   // UNICODE_TO_GBK[10710] := 16#601E;
   // UNICODE_TO_GBK[10711] := 16#904A;
   // UNICODE_TO_GBK[10712] := 16#601F;
   // UNICODE_TO_GBK[10713] := 16#904B;
   // UNICODE_TO_GBK[10714] := 16#6020;
   // UNICODE_TO_GBK[10715] := 16#B5A1;
   // UNICODE_TO_GBK[10716] := 16#6021;
   // UNICODE_TO_GBK[10717] := 16#E2F9;
   // UNICODE_TO_GBK[10718] := 16#6022;
   // UNICODE_TO_GBK[10719] := 16#904C;
   // UNICODE_TO_GBK[10720] := 16#6023;
   // UNICODE_TO_GBK[10721] := 16#904D;
   // UNICODE_TO_GBK[10722] := 16#6024;
   // UNICODE_TO_GBK[10723] := 16#904E;
   // UNICODE_TO_GBK[10724] := 16#6025;
   // UNICODE_TO_GBK[10725] := 16#BCB1;
   // UNICODE_TO_GBK[10726] := 16#6026;
   // UNICODE_TO_GBK[10727] := 16#E2F1;
   // UNICODE_TO_GBK[10728] := 16#6027;
   // UNICODE_TO_GBK[10729] := 16#D0D4;
   // UNICODE_TO_GBK[10730] := 16#6028;
   // UNICODE_TO_GBK[10731] := 16#D4B9;
   // UNICODE_TO_GBK[10732] := 16#6029;
   // UNICODE_TO_GBK[10733] := 16#E2F5;
   // UNICODE_TO_GBK[10734] := 16#602A;
   // UNICODE_TO_GBK[10735] := 16#B9D6;
   // UNICODE_TO_GBK[10736] := 16#602B;
   // UNICODE_TO_GBK[10737] := 16#E2F6;
   // UNICODE_TO_GBK[10738] := 16#602C;
   // UNICODE_TO_GBK[10739] := 16#904F;
   // UNICODE_TO_GBK[10740] := 16#602D;
   // UNICODE_TO_GBK[10741] := 16#9050;
   // UNICODE_TO_GBK[10742] := 16#602E;
   // UNICODE_TO_GBK[10743] := 16#9051;
   // UNICODE_TO_GBK[10744] := 16#602F;
   // UNICODE_TO_GBK[10745] := 16#C7D3;
   // UNICODE_TO_GBK[10746] := 16#6030;
   // UNICODE_TO_GBK[10747] := 16#9052;
   // UNICODE_TO_GBK[10748] := 16#6031;
   // UNICODE_TO_GBK[10749] := 16#9053;
   // UNICODE_TO_GBK[10750] := 16#6032;
   // UNICODE_TO_GBK[10751] := 16#9054;
   // UNICODE_TO_GBK[10752] := 16#6033;
   // UNICODE_TO_GBK[10753] := 16#9055;
   // UNICODE_TO_GBK[10754] := 16#6034;
   // UNICODE_TO_GBK[10755] := 16#9056;
   // UNICODE_TO_GBK[10756] := 16#6035;
   // UNICODE_TO_GBK[10757] := 16#E2F0;
   // UNICODE_TO_GBK[10758] := 16#6036;
   // UNICODE_TO_GBK[10759] := 16#9057;
   // UNICODE_TO_GBK[10760] := 16#6037;
   // UNICODE_TO_GBK[10761] := 16#9058;
   // UNICODE_TO_GBK[10762] := 16#6038;
   // UNICODE_TO_GBK[10763] := 16#9059;
   // UNICODE_TO_GBK[10764] := 16#6039;
   // UNICODE_TO_GBK[10765] := 16#905A;
   // UNICODE_TO_GBK[10766] := 16#603A;
   // UNICODE_TO_GBK[10767] := 16#905B;
   // UNICODE_TO_GBK[10768] := 16#603B;
   // UNICODE_TO_GBK[10769] := 16#D7DC;
   // UNICODE_TO_GBK[10770] := 16#603C;
   // UNICODE_TO_GBK[10771] := 16#EDA1;
   // UNICODE_TO_GBK[10772] := 16#603D;
   // UNICODE_TO_GBK[10773] := 16#905C;
   // UNICODE_TO_GBK[10774] := 16#603E;
   // UNICODE_TO_GBK[10775] := 16#905D;
   // UNICODE_TO_GBK[10776] := 16#603F;
   // UNICODE_TO_GBK[10777] := 16#E2F8;
   // UNICODE_TO_GBK[10778] := 16#6040;
   // UNICODE_TO_GBK[10779] := 16#905E;
   // UNICODE_TO_GBK[10780] := 16#6041;
   // UNICODE_TO_GBK[10781] := 16#EDA5;
   // UNICODE_TO_GBK[10782] := 16#6042;
   // UNICODE_TO_GBK[10783] := 16#E2FE;
   // UNICODE_TO_GBK[10784] := 16#6043;
   // UNICODE_TO_GBK[10785] := 16#CAD1;
   // UNICODE_TO_GBK[10786] := 16#6044;
   // UNICODE_TO_GBK[10787] := 16#905F;
   // UNICODE_TO_GBK[10788] := 16#6045;
   // UNICODE_TO_GBK[10789] := 16#9060;
   // UNICODE_TO_GBK[10790] := 16#6046;
   // UNICODE_TO_GBK[10791] := 16#9061;
   // UNICODE_TO_GBK[10792] := 16#6047;
   // UNICODE_TO_GBK[10793] := 16#9062;
   // UNICODE_TO_GBK[10794] := 16#6048;
   // UNICODE_TO_GBK[10795] := 16#9063;
   // UNICODE_TO_GBK[10796] := 16#6049;
   // UNICODE_TO_GBK[10797] := 16#9064;
   // UNICODE_TO_GBK[10798] := 16#604A;
   // UNICODE_TO_GBK[10799] := 16#9065;
   // UNICODE_TO_GBK[10800] := 16#604B;
   // UNICODE_TO_GBK[10801] := 16#C1B5;
   // UNICODE_TO_GBK[10802] := 16#604C;
   // UNICODE_TO_GBK[10803] := 16#9066;
   // UNICODE_TO_GBK[10804] := 16#604D;
   // UNICODE_TO_GBK[10805] := 16#BBD0;
   // UNICODE_TO_GBK[10806] := 16#604E;
   // UNICODE_TO_GBK[10807] := 16#9067;
   // UNICODE_TO_GBK[10808] := 16#604F;
   // UNICODE_TO_GBK[10809] := 16#9068;
   // UNICODE_TO_GBK[10810] := 16#6050;
   // UNICODE_TO_GBK[10811] := 16#BFD6;
   // UNICODE_TO_GBK[10812] := 16#6051;
   // UNICODE_TO_GBK[10813] := 16#9069;
   // UNICODE_TO_GBK[10814] := 16#6052;
   // UNICODE_TO_GBK[10815] := 16#BAE3;
   // UNICODE_TO_GBK[10816] := 16#6053;
   // UNICODE_TO_GBK[10817] := 16#906A;
   // UNICODE_TO_GBK[10818] := 16#6054;
   // UNICODE_TO_GBK[10819] := 16#906B;
   // UNICODE_TO_GBK[10820] := 16#6055;
   // UNICODE_TO_GBK[10821] := 16#CBA1;
   // UNICODE_TO_GBK[10822] := 16#6056;
   // UNICODE_TO_GBK[10823] := 16#906C;
   // UNICODE_TO_GBK[10824] := 16#6057;
   // UNICODE_TO_GBK[10825] := 16#906D;
   // UNICODE_TO_GBK[10826] := 16#6058;
   // UNICODE_TO_GBK[10827] := 16#906E;
   // UNICODE_TO_GBK[10828] := 16#6059;
   // UNICODE_TO_GBK[10829] := 16#EDA6;
   // UNICODE_TO_GBK[10830] := 16#605A;
   // UNICODE_TO_GBK[10831] := 16#EDA3;
   // UNICODE_TO_GBK[10832] := 16#605B;
   // UNICODE_TO_GBK[10833] := 16#906F;
   // UNICODE_TO_GBK[10834] := 16#605C;
   // UNICODE_TO_GBK[10835] := 16#9070;
   // UNICODE_TO_GBK[10836] := 16#605D;
   // UNICODE_TO_GBK[10837] := 16#EDA2;
   // UNICODE_TO_GBK[10838] := 16#605E;
   // UNICODE_TO_GBK[10839] := 16#9071;
   // UNICODE_TO_GBK[10840] := 16#605F;
   // UNICODE_TO_GBK[10841] := 16#9072;
   // UNICODE_TO_GBK[10842] := 16#6060;
   // UNICODE_TO_GBK[10843] := 16#9073;
   // UNICODE_TO_GBK[10844] := 16#6061;
   // UNICODE_TO_GBK[10845] := 16#9074;
   // UNICODE_TO_GBK[10846] := 16#6062;
   // UNICODE_TO_GBK[10847] := 16#BBD6;
   // UNICODE_TO_GBK[10848] := 16#6063;
   // UNICODE_TO_GBK[10849] := 16#EDA7;
   // UNICODE_TO_GBK[10850] := 16#6064;
   // UNICODE_TO_GBK[10851] := 16#D0F4;
   // UNICODE_TO_GBK[10852] := 16#6065;
   // UNICODE_TO_GBK[10853] := 16#9075;
   // UNICODE_TO_GBK[10854] := 16#6066;
   // UNICODE_TO_GBK[10855] := 16#9076;
   // UNICODE_TO_GBK[10856] := 16#6067;
   // UNICODE_TO_GBK[10857] := 16#EDA4;
   // UNICODE_TO_GBK[10858] := 16#6068;
   // UNICODE_TO_GBK[10859] := 16#BADE;
   // UNICODE_TO_GBK[10860] := 16#6069;
   // UNICODE_TO_GBK[10861] := 16#B6F7;
   // UNICODE_TO_GBK[10862] := 16#606A;
   // UNICODE_TO_GBK[10863] := 16#E3A1;
   // UNICODE_TO_GBK[10864] := 16#606B;
   // UNICODE_TO_GBK[10865] := 16#B6B2;
   // UNICODE_TO_GBK[10866] := 16#606C;
   // UNICODE_TO_GBK[10867] := 16#CCF1;
   // UNICODE_TO_GBK[10868] := 16#606D;
   // UNICODE_TO_GBK[10869] := 16#B9A7;
   // UNICODE_TO_GBK[10870] := 16#606E;
   // UNICODE_TO_GBK[10871] := 16#9077;
   // UNICODE_TO_GBK[10872] := 16#606F;
   // UNICODE_TO_GBK[10873] := 16#CFA2;
   // UNICODE_TO_GBK[10874] := 16#6070;
   // UNICODE_TO_GBK[10875] := 16#C7A1;
   // UNICODE_TO_GBK[10876] := 16#6071;
   // UNICODE_TO_GBK[10877] := 16#9078;
   // UNICODE_TO_GBK[10878] := 16#6072;
   // UNICODE_TO_GBK[10879] := 16#9079;
   // UNICODE_TO_GBK[10880] := 16#6073;
   // UNICODE_TO_GBK[10881] := 16#BFD2;
   // UNICODE_TO_GBK[10882] := 16#6074;
   // UNICODE_TO_GBK[10883] := 16#907A;
   // UNICODE_TO_GBK[10884] := 16#6075;
   // UNICODE_TO_GBK[10885] := 16#907B;
   // UNICODE_TO_GBK[10886] := 16#6076;
   // UNICODE_TO_GBK[10887] := 16#B6F1;
   // UNICODE_TO_GBK[10888] := 16#6077;
   // UNICODE_TO_GBK[10889] := 16#907C;
   // UNICODE_TO_GBK[10890] := 16#6078;
   // UNICODE_TO_GBK[10891] := 16#E2FA;
   // UNICODE_TO_GBK[10892] := 16#6079;
   // UNICODE_TO_GBK[10893] := 16#E2FB;
   // UNICODE_TO_GBK[10894] := 16#607A;
   // UNICODE_TO_GBK[10895] := 16#E2FD;
   // UNICODE_TO_GBK[10896] := 16#607B;
   // UNICODE_TO_GBK[10897] := 16#E2FC;
   // UNICODE_TO_GBK[10898] := 16#607C;
   // UNICODE_TO_GBK[10899] := 16#C4D5;
   // UNICODE_TO_GBK[10900] := 16#607D;
   // UNICODE_TO_GBK[10901] := 16#E3A2;
   // UNICODE_TO_GBK[10902] := 16#607E;
   // UNICODE_TO_GBK[10903] := 16#907D;
   // UNICODE_TO_GBK[10904] := 16#607F;
   // UNICODE_TO_GBK[10905] := 16#D3C1;
   // UNICODE_TO_GBK[10906] := 16#6080;
   // UNICODE_TO_GBK[10907] := 16#907E;
   // UNICODE_TO_GBK[10908] := 16#6081;
   // UNICODE_TO_GBK[10909] := 16#9080;
   // UNICODE_TO_GBK[10910] := 16#6082;
   // UNICODE_TO_GBK[10911] := 16#9081;
   // UNICODE_TO_GBK[10912] := 16#6083;
   // UNICODE_TO_GBK[10913] := 16#E3A7;
   // UNICODE_TO_GBK[10914] := 16#6084;
   // UNICODE_TO_GBK[10915] := 16#C7C4;
   // UNICODE_TO_GBK[10916] := 16#6085;
   // UNICODE_TO_GBK[10917] := 16#9082;
   // UNICODE_TO_GBK[10918] := 16#6086;
   // UNICODE_TO_GBK[10919] := 16#9083;
   // UNICODE_TO_GBK[10920] := 16#6087;
   // UNICODE_TO_GBK[10921] := 16#9084;
   // UNICODE_TO_GBK[10922] := 16#6088;
   // UNICODE_TO_GBK[10923] := 16#9085;
   // UNICODE_TO_GBK[10924] := 16#6089;
   // UNICODE_TO_GBK[10925] := 16#CFA4;
   // UNICODE_TO_GBK[10926] := 16#608A;
   // UNICODE_TO_GBK[10927] := 16#9086;
   // UNICODE_TO_GBK[10928] := 16#608B;
   // UNICODE_TO_GBK[10929] := 16#9087;
   // UNICODE_TO_GBK[10930] := 16#608C;
   // UNICODE_TO_GBK[10931] := 16#E3A9;
   // UNICODE_TO_GBK[10932] := 16#608D;
   // UNICODE_TO_GBK[10933] := 16#BAB7;
   // UNICODE_TO_GBK[10934] := 16#608E;
   // UNICODE_TO_GBK[10935] := 16#9088;
   // UNICODE_TO_GBK[10936] := 16#608F;
   // UNICODE_TO_GBK[10937] := 16#9089;
   // UNICODE_TO_GBK[10938] := 16#6090;
   // UNICODE_TO_GBK[10939] := 16#908A;
   // UNICODE_TO_GBK[10940] := 16#6091;
   // UNICODE_TO_GBK[10941] := 16#908B;
   // UNICODE_TO_GBK[10942] := 16#6092;
   // UNICODE_TO_GBK[10943] := 16#E3A8;
   // UNICODE_TO_GBK[10944] := 16#6093;
   // UNICODE_TO_GBK[10945] := 16#908C;
   // UNICODE_TO_GBK[10946] := 16#6094;
   // UNICODE_TO_GBK[10947] := 16#BBDA;
   // UNICODE_TO_GBK[10948] := 16#6095;
   // UNICODE_TO_GBK[10949] := 16#908D;
   // UNICODE_TO_GBK[10950] := 16#6096;
   // UNICODE_TO_GBK[10951] := 16#E3A3;
   // UNICODE_TO_GBK[10952] := 16#6097;
   // UNICODE_TO_GBK[10953] := 16#908E;
   // UNICODE_TO_GBK[10954] := 16#6098;
   // UNICODE_TO_GBK[10955] := 16#908F;
   // UNICODE_TO_GBK[10956] := 16#6099;
   // UNICODE_TO_GBK[10957] := 16#9090;
   // UNICODE_TO_GBK[10958] := 16#609A;
   // UNICODE_TO_GBK[10959] := 16#E3A4;
   // UNICODE_TO_GBK[10960] := 16#609B;
   // UNICODE_TO_GBK[10961] := 16#E3AA;
   // UNICODE_TO_GBK[10962] := 16#609C;
   // UNICODE_TO_GBK[10963] := 16#9091;
   // UNICODE_TO_GBK[10964] := 16#609D;
   // UNICODE_TO_GBK[10965] := 16#E3A6;
   // UNICODE_TO_GBK[10966] := 16#609E;
   // UNICODE_TO_GBK[10967] := 16#9092;
   // UNICODE_TO_GBK[10968] := 16#609F;
   // UNICODE_TO_GBK[10969] := 16#CEF2;
   // UNICODE_TO_GBK[10970] := 16#60A0;
   // UNICODE_TO_GBK[10971] := 16#D3C6;
   // UNICODE_TO_GBK[10972] := 16#60A1;
   // UNICODE_TO_GBK[10973] := 16#9093;
   // UNICODE_TO_GBK[10974] := 16#60A2;
   // UNICODE_TO_GBK[10975] := 16#9094;
   // UNICODE_TO_GBK[10976] := 16#60A3;
   // UNICODE_TO_GBK[10977] := 16#BBBC;
   // UNICODE_TO_GBK[10978] := 16#60A4;
   // UNICODE_TO_GBK[10979] := 16#9095;
   // UNICODE_TO_GBK[10980] := 16#60A5;
   // UNICODE_TO_GBK[10981] := 16#9096;
   // UNICODE_TO_GBK[10982] := 16#60A6;
   // UNICODE_TO_GBK[10983] := 16#D4C3;
   // UNICODE_TO_GBK[10984] := 16#60A7;
   // UNICODE_TO_GBK[10985] := 16#9097;
   // UNICODE_TO_GBK[10986] := 16#60A8;
   // UNICODE_TO_GBK[10987] := 16#C4FA;
   // UNICODE_TO_GBK[10988] := 16#60A9;
   // UNICODE_TO_GBK[10989] := 16#9098;
   // UNICODE_TO_GBK[10990] := 16#60AA;
   // UNICODE_TO_GBK[10991] := 16#9099;
   // UNICODE_TO_GBK[10992] := 16#60AB;
   // UNICODE_TO_GBK[10993] := 16#EDA8;
   // UNICODE_TO_GBK[10994] := 16#60AC;
   // UNICODE_TO_GBK[10995] := 16#D0FC;
   // UNICODE_TO_GBK[10996] := 16#60AD;
   // UNICODE_TO_GBK[10997] := 16#E3A5;
   // UNICODE_TO_GBK[10998] := 16#60AE;
   // UNICODE_TO_GBK[10999] := 16#909A;
   // UNICODE_TO_GBK[11000] := 16#60AF;
   // UNICODE_TO_GBK[11001] := 16#C3F5;
   // UNICODE_TO_GBK[11002] := 16#60B0;
   // UNICODE_TO_GBK[11003] := 16#909B;
   // UNICODE_TO_GBK[11004] := 16#60B1;
   // UNICODE_TO_GBK[11005] := 16#E3AD;
   // UNICODE_TO_GBK[11006] := 16#60B2;
   // UNICODE_TO_GBK[11007] := 16#B1AF;
   // UNICODE_TO_GBK[11008] := 16#60B3;
   // UNICODE_TO_GBK[11009] := 16#909C;
   // UNICODE_TO_GBK[11010] := 16#60B4;
   // UNICODE_TO_GBK[11011] := 16#E3B2;
   // UNICODE_TO_GBK[11012] := 16#60B5;
   // UNICODE_TO_GBK[11013] := 16#909D;
   // UNICODE_TO_GBK[11014] := 16#60B6;
   // UNICODE_TO_GBK[11015] := 16#909E;
   // UNICODE_TO_GBK[11016] := 16#60B7;
   // UNICODE_TO_GBK[11017] := 16#909F;
   // UNICODE_TO_GBK[11018] := 16#60B8;
   // UNICODE_TO_GBK[11019] := 16#BCC2;
   // UNICODE_TO_GBK[11020] := 16#60B9;
   // UNICODE_TO_GBK[11021] := 16#90A0;
   // UNICODE_TO_GBK[11022] := 16#60BA;
   // UNICODE_TO_GBK[11023] := 16#90A1;
   // UNICODE_TO_GBK[11024] := 16#60BB;
   // UNICODE_TO_GBK[11025] := 16#E3AC;
   // UNICODE_TO_GBK[11026] := 16#60BC;
   // UNICODE_TO_GBK[11027] := 16#B5BF;
   // UNICODE_TO_GBK[11028] := 16#60BD;
   // UNICODE_TO_GBK[11029] := 16#90A2;
   // UNICODE_TO_GBK[11030] := 16#60BE;
   // UNICODE_TO_GBK[11031] := 16#90A3;
   // UNICODE_TO_GBK[11032] := 16#60BF;
   // UNICODE_TO_GBK[11033] := 16#90A4;
   // UNICODE_TO_GBK[11034] := 16#60C0;
   // UNICODE_TO_GBK[11035] := 16#90A5;
   // UNICODE_TO_GBK[11036] := 16#60C1;
   // UNICODE_TO_GBK[11037] := 16#90A6;
   // UNICODE_TO_GBK[11038] := 16#60C2;
   // UNICODE_TO_GBK[11039] := 16#90A7;
   // UNICODE_TO_GBK[11040] := 16#60C3;
   // UNICODE_TO_GBK[11041] := 16#90A8;
   // UNICODE_TO_GBK[11042] := 16#60C4;
   // UNICODE_TO_GBK[11043] := 16#90A9;
   // UNICODE_TO_GBK[11044] := 16#60C5;
   // UNICODE_TO_GBK[11045] := 16#C7E9;
   // UNICODE_TO_GBK[11046] := 16#60C6;
   // UNICODE_TO_GBK[11047] := 16#E3B0;
   // UNICODE_TO_GBK[11048] := 16#60C7;
   // UNICODE_TO_GBK[11049] := 16#90AA;
   // UNICODE_TO_GBK[11050] := 16#60C8;
   // UNICODE_TO_GBK[11051] := 16#90AB;
   // UNICODE_TO_GBK[11052] := 16#60C9;
   // UNICODE_TO_GBK[11053] := 16#90AC;
   // UNICODE_TO_GBK[11054] := 16#60CA;
   // UNICODE_TO_GBK[11055] := 16#BEAA;
   // UNICODE_TO_GBK[11056] := 16#60CB;
   // UNICODE_TO_GBK[11057] := 16#CDEF;
   // UNICODE_TO_GBK[11058] := 16#60CC;
   // UNICODE_TO_GBK[11059] := 16#90AD;
   // UNICODE_TO_GBK[11060] := 16#60CD;
   // UNICODE_TO_GBK[11061] := 16#90AE;
   // UNICODE_TO_GBK[11062] := 16#60CE;
   // UNICODE_TO_GBK[11063] := 16#90AF;
   // UNICODE_TO_GBK[11064] := 16#60CF;
   // UNICODE_TO_GBK[11065] := 16#90B0;
   // UNICODE_TO_GBK[11066] := 16#60D0;
   // UNICODE_TO_GBK[11067] := 16#90B1;
   // UNICODE_TO_GBK[11068] := 16#60D1;
   // UNICODE_TO_GBK[11069] := 16#BBF3;
   // UNICODE_TO_GBK[11070] := 16#60D2;
   // UNICODE_TO_GBK[11071] := 16#90B2;
   // UNICODE_TO_GBK[11072] := 16#60D3;
   // UNICODE_TO_GBK[11073] := 16#90B3;
   // UNICODE_TO_GBK[11074] := 16#60D4;
   // UNICODE_TO_GBK[11075] := 16#90B4;
   // UNICODE_TO_GBK[11076] := 16#60D5;
   // UNICODE_TO_GBK[11077] := 16#CCE8;
   // UNICODE_TO_GBK[11078] := 16#60D6;
   // UNICODE_TO_GBK[11079] := 16#90B5;
   // UNICODE_TO_GBK[11080] := 16#60D7;
   // UNICODE_TO_GBK[11081] := 16#90B6;
   // UNICODE_TO_GBK[11082] := 16#60D8;
   // UNICODE_TO_GBK[11083] := 16#E3AF;
   // UNICODE_TO_GBK[11084] := 16#60D9;
   // UNICODE_TO_GBK[11085] := 16#90B7;
   // UNICODE_TO_GBK[11086] := 16#60DA;
   // UNICODE_TO_GBK[11087] := 16#E3B1;
   // UNICODE_TO_GBK[11088] := 16#60DB;
   // UNICODE_TO_GBK[11089] := 16#90B8;
   // UNICODE_TO_GBK[11090] := 16#60DC;
   // UNICODE_TO_GBK[11091] := 16#CFA7;
   // UNICODE_TO_GBK[11092] := 16#60DD;
   // UNICODE_TO_GBK[11093] := 16#E3AE;
   // UNICODE_TO_GBK[11094] := 16#60DE;
   // UNICODE_TO_GBK[11095] := 16#90B9;
   // UNICODE_TO_GBK[11096] := 16#60DF;
   // UNICODE_TO_GBK[11097] := 16#CEA9;
   // UNICODE_TO_GBK[11098] := 16#60E0;
   // UNICODE_TO_GBK[11099] := 16#BBDD;
   // UNICODE_TO_GBK[11100] := 16#60E1;
   // UNICODE_TO_GBK[11101] := 16#90BA;
   // UNICODE_TO_GBK[11102] := 16#60E2;
   // UNICODE_TO_GBK[11103] := 16#90BB;
   // UNICODE_TO_GBK[11104] := 16#60E3;
   // UNICODE_TO_GBK[11105] := 16#90BC;
   // UNICODE_TO_GBK[11106] := 16#60E4;
   // UNICODE_TO_GBK[11107] := 16#90BD;
   // UNICODE_TO_GBK[11108] := 16#60E5;
   // UNICODE_TO_GBK[11109] := 16#90BE;
   // UNICODE_TO_GBK[11110] := 16#60E6;
   // UNICODE_TO_GBK[11111] := 16#B5EB;
   // UNICODE_TO_GBK[11112] := 16#60E7;
   // UNICODE_TO_GBK[11113] := 16#BEE5;
   // UNICODE_TO_GBK[11114] := 16#60E8;
   // UNICODE_TO_GBK[11115] := 16#B2D2;
   // UNICODE_TO_GBK[11116] := 16#60E9;
   // UNICODE_TO_GBK[11117] := 16#B3CD;
   // UNICODE_TO_GBK[11118] := 16#60EA;
   // UNICODE_TO_GBK[11119] := 16#90BF;
   // UNICODE_TO_GBK[11120] := 16#60EB;
   // UNICODE_TO_GBK[11121] := 16#B1B9;
   // UNICODE_TO_GBK[11122] := 16#60EC;
   // UNICODE_TO_GBK[11123] := 16#E3AB;
   // UNICODE_TO_GBK[11124] := 16#60ED;
   // UNICODE_TO_GBK[11125] := 16#B2D1;
   // UNICODE_TO_GBK[11126] := 16#60EE;
   // UNICODE_TO_GBK[11127] := 16#B5AC;
   // UNICODE_TO_GBK[11128] := 16#60EF;
   // UNICODE_TO_GBK[11129] := 16#B9DF;
   // UNICODE_TO_GBK[11130] := 16#60F0;
   // UNICODE_TO_GBK[11131] := 16#B6E8;
   // UNICODE_TO_GBK[11132] := 16#60F1;
   // UNICODE_TO_GBK[11133] := 16#90C0;
   // UNICODE_TO_GBK[11134] := 16#60F2;
   // UNICODE_TO_GBK[11135] := 16#90C1;
   // UNICODE_TO_GBK[11136] := 16#60F3;
   // UNICODE_TO_GBK[11137] := 16#CFEB;
   // UNICODE_TO_GBK[11138] := 16#60F4;
   // UNICODE_TO_GBK[11139] := 16#E3B7;
   // UNICODE_TO_GBK[11140] := 16#60F5;
   // UNICODE_TO_GBK[11141] := 16#90C2;
   // UNICODE_TO_GBK[11142] := 16#60F6;
   // UNICODE_TO_GBK[11143] := 16#BBCC;
   // UNICODE_TO_GBK[11144] := 16#60F7;
   // UNICODE_TO_GBK[11145] := 16#90C3;
   // UNICODE_TO_GBK[11146] := 16#60F8;
   // UNICODE_TO_GBK[11147] := 16#90C4;
   // UNICODE_TO_GBK[11148] := 16#60F9;
   // UNICODE_TO_GBK[11149] := 16#C8C7;
   // UNICODE_TO_GBK[11150] := 16#60FA;
   // UNICODE_TO_GBK[11151] := 16#D0CA;
   // UNICODE_TO_GBK[11152] := 16#60FB;
   // UNICODE_TO_GBK[11153] := 16#90C5;
   // UNICODE_TO_GBK[11154] := 16#60FC;
   // UNICODE_TO_GBK[11155] := 16#90C6;
   // UNICODE_TO_GBK[11156] := 16#60FD;
   // UNICODE_TO_GBK[11157] := 16#90C7;
   // UNICODE_TO_GBK[11158] := 16#60FE;
   // UNICODE_TO_GBK[11159] := 16#90C8;
   // UNICODE_TO_GBK[11160] := 16#60FF;
   // UNICODE_TO_GBK[11161] := 16#90C9;
   // UNICODE_TO_GBK[11162] := 16#6100;
   // UNICODE_TO_GBK[11163] := 16#E3B8;
   // UNICODE_TO_GBK[11164] := 16#6101;
   // UNICODE_TO_GBK[11165] := 16#B3EE;
   // UNICODE_TO_GBK[11166] := 16#6102;
   // UNICODE_TO_GBK[11167] := 16#90CA;
   // UNICODE_TO_GBK[11168] := 16#6103;
   // UNICODE_TO_GBK[11169] := 16#90CB;
   // UNICODE_TO_GBK[11170] := 16#6104;
   // UNICODE_TO_GBK[11171] := 16#90CC;
   // UNICODE_TO_GBK[11172] := 16#6105;
   // UNICODE_TO_GBK[11173] := 16#90CD;
   // UNICODE_TO_GBK[11174] := 16#6106;
   // UNICODE_TO_GBK[11175] := 16#EDA9;
   // UNICODE_TO_GBK[11176] := 16#6107;
   // UNICODE_TO_GBK[11177] := 16#90CE;
   // UNICODE_TO_GBK[11178] := 16#6108;
   // UNICODE_TO_GBK[11179] := 16#D3FA;
   // UNICODE_TO_GBK[11180] := 16#6109;
   // UNICODE_TO_GBK[11181] := 16#D3E4;
   // UNICODE_TO_GBK[11182] := 16#610A;
   // UNICODE_TO_GBK[11183] := 16#90CF;
   // UNICODE_TO_GBK[11184] := 16#610B;
   // UNICODE_TO_GBK[11185] := 16#90D0;
   // UNICODE_TO_GBK[11186] := 16#610C;
   // UNICODE_TO_GBK[11187] := 16#90D1;
   // UNICODE_TO_GBK[11188] := 16#610D;
   // UNICODE_TO_GBK[11189] := 16#EDAA;
   // UNICODE_TO_GBK[11190] := 16#610E;
   // UNICODE_TO_GBK[11191] := 16#E3B9;
   // UNICODE_TO_GBK[11192] := 16#610F;
   // UNICODE_TO_GBK[11193] := 16#D2E2;
   // UNICODE_TO_GBK[11194] := 16#6110;
   // UNICODE_TO_GBK[11195] := 16#90D2;
   // UNICODE_TO_GBK[11196] := 16#6111;
   // UNICODE_TO_GBK[11197] := 16#90D3;
   // UNICODE_TO_GBK[11198] := 16#6112;
   // UNICODE_TO_GBK[11199] := 16#90D4;
   // UNICODE_TO_GBK[11200] := 16#6113;
   // UNICODE_TO_GBK[11201] := 16#90D5;
   // UNICODE_TO_GBK[11202] := 16#6114;
   // UNICODE_TO_GBK[11203] := 16#90D6;
   // UNICODE_TO_GBK[11204] := 16#6115;
   // UNICODE_TO_GBK[11205] := 16#E3B5;
   // UNICODE_TO_GBK[11206] := 16#6116;
   // UNICODE_TO_GBK[11207] := 16#90D7;
   // UNICODE_TO_GBK[11208] := 16#6117;
   // UNICODE_TO_GBK[11209] := 16#90D8;
   // UNICODE_TO_GBK[11210] := 16#6118;
   // UNICODE_TO_GBK[11211] := 16#90D9;
   // UNICODE_TO_GBK[11212] := 16#6119;
   // UNICODE_TO_GBK[11213] := 16#90DA;
   // UNICODE_TO_GBK[11214] := 16#611A;
   // UNICODE_TO_GBK[11215] := 16#D3DE;
   // UNICODE_TO_GBK[11216] := 16#611B;
   // UNICODE_TO_GBK[11217] := 16#90DB;
   // UNICODE_TO_GBK[11218] := 16#611C;
   // UNICODE_TO_GBK[11219] := 16#90DC;
   // UNICODE_TO_GBK[11220] := 16#611D;
   // UNICODE_TO_GBK[11221] := 16#90DD;
   // UNICODE_TO_GBK[11222] := 16#611E;
   // UNICODE_TO_GBK[11223] := 16#90DE;
   // UNICODE_TO_GBK[11224] := 16#611F;
   // UNICODE_TO_GBK[11225] := 16#B8D0;
   // UNICODE_TO_GBK[11226] := 16#6120;
   // UNICODE_TO_GBK[11227] := 16#E3B3;
   // UNICODE_TO_GBK[11228] := 16#6121;
   // UNICODE_TO_GBK[11229] := 16#90DF;
   // UNICODE_TO_GBK[11230] := 16#6122;
   // UNICODE_TO_GBK[11231] := 16#90E0;
   // UNICODE_TO_GBK[11232] := 16#6123;
   // UNICODE_TO_GBK[11233] := 16#E3B6;
   // UNICODE_TO_GBK[11234] := 16#6124;
   // UNICODE_TO_GBK[11235] := 16#B7DF;
   // UNICODE_TO_GBK[11236] := 16#6125;
   // UNICODE_TO_GBK[11237] := 16#90E1;
   // UNICODE_TO_GBK[11238] := 16#6126;
   // UNICODE_TO_GBK[11239] := 16#E3B4;
   // UNICODE_TO_GBK[11240] := 16#6127;
   // UNICODE_TO_GBK[11241] := 16#C0A2;
   // UNICODE_TO_GBK[11242] := 16#6128;
   // UNICODE_TO_GBK[11243] := 16#90E2;
   // UNICODE_TO_GBK[11244] := 16#6129;
   // UNICODE_TO_GBK[11245] := 16#90E3;
   // UNICODE_TO_GBK[11246] := 16#612A;
   // UNICODE_TO_GBK[11247] := 16#90E4;
   // UNICODE_TO_GBK[11248] := 16#612B;
   // UNICODE_TO_GBK[11249] := 16#E3BA;
   // UNICODE_TO_GBK[11250] := 16#612C;
   // UNICODE_TO_GBK[11251] := 16#90E5;
   // UNICODE_TO_GBK[11252] := 16#612D;
   // UNICODE_TO_GBK[11253] := 16#90E6;
   // UNICODE_TO_GBK[11254] := 16#612E;
   // UNICODE_TO_GBK[11255] := 16#90E7;
   // UNICODE_TO_GBK[11256] := 16#612F;
   // UNICODE_TO_GBK[11257] := 16#90E8;
   // UNICODE_TO_GBK[11258] := 16#6130;
   // UNICODE_TO_GBK[11259] := 16#90E9;
   // UNICODE_TO_GBK[11260] := 16#6131;
   // UNICODE_TO_GBK[11261] := 16#90EA;
   // UNICODE_TO_GBK[11262] := 16#6132;
   // UNICODE_TO_GBK[11263] := 16#90EB;
   // UNICODE_TO_GBK[11264] := 16#6133;
   // UNICODE_TO_GBK[11265] := 16#90EC;
   // UNICODE_TO_GBK[11266] := 16#6134;
   // UNICODE_TO_GBK[11267] := 16#90ED;
   // UNICODE_TO_GBK[11268] := 16#6135;
   // UNICODE_TO_GBK[11269] := 16#90EE;
   // UNICODE_TO_GBK[11270] := 16#6136;
   // UNICODE_TO_GBK[11271] := 16#90EF;
   // UNICODE_TO_GBK[11272] := 16#6137;
   // UNICODE_TO_GBK[11273] := 16#90F0;
   // UNICODE_TO_GBK[11274] := 16#6138;
   // UNICODE_TO_GBK[11275] := 16#90F1;
   // UNICODE_TO_GBK[11276] := 16#6139;
   // UNICODE_TO_GBK[11277] := 16#90F2;
   // UNICODE_TO_GBK[11278] := 16#613A;
   // UNICODE_TO_GBK[11279] := 16#90F3;
   // UNICODE_TO_GBK[11280] := 16#613B;
   // UNICODE_TO_GBK[11281] := 16#90F4;
   // UNICODE_TO_GBK[11282] := 16#613C;
   // UNICODE_TO_GBK[11283] := 16#90F5;
   // UNICODE_TO_GBK[11284] := 16#613D;
   // UNICODE_TO_GBK[11285] := 16#90F6;
   // UNICODE_TO_GBK[11286] := 16#613E;
   // UNICODE_TO_GBK[11287] := 16#90F7;
   // UNICODE_TO_GBK[11288] := 16#613F;
   // UNICODE_TO_GBK[11289] := 16#D4B8;
   // UNICODE_TO_GBK[11290] := 16#6140;
   // UNICODE_TO_GBK[11291] := 16#90F8;
   // UNICODE_TO_GBK[11292] := 16#6141;
   // UNICODE_TO_GBK[11293] := 16#90F9;
   // UNICODE_TO_GBK[11294] := 16#6142;
   // UNICODE_TO_GBK[11295] := 16#90FA;
   // UNICODE_TO_GBK[11296] := 16#6143;
   // UNICODE_TO_GBK[11297] := 16#90FB;
   // UNICODE_TO_GBK[11298] := 16#6144;
   // UNICODE_TO_GBK[11299] := 16#90FC;
   // UNICODE_TO_GBK[11300] := 16#6145;
   // UNICODE_TO_GBK[11301] := 16#90FD;
   // UNICODE_TO_GBK[11302] := 16#6146;
   // UNICODE_TO_GBK[11303] := 16#90FE;
   // UNICODE_TO_GBK[11304] := 16#6147;
   // UNICODE_TO_GBK[11305] := 16#9140;
   // UNICODE_TO_GBK[11306] := 16#6148;
   // UNICODE_TO_GBK[11307] := 16#B4C8;
   // UNICODE_TO_GBK[11308] := 16#6149;
   // UNICODE_TO_GBK[11309] := 16#9141;
   // UNICODE_TO_GBK[11310] := 16#614A;
   // UNICODE_TO_GBK[11311] := 16#E3BB;
   // UNICODE_TO_GBK[11312] := 16#614B;
   // UNICODE_TO_GBK[11313] := 16#9142;
   // UNICODE_TO_GBK[11314] := 16#614C;
   // UNICODE_TO_GBK[11315] := 16#BBC5;
   // UNICODE_TO_GBK[11316] := 16#614D;
   // UNICODE_TO_GBK[11317] := 16#9143;
   // UNICODE_TO_GBK[11318] := 16#614E;
   // UNICODE_TO_GBK[11319] := 16#C9F7;
   // UNICODE_TO_GBK[11320] := 16#614F;
   // UNICODE_TO_GBK[11321] := 16#9144;
   // UNICODE_TO_GBK[11322] := 16#6150;
   // UNICODE_TO_GBK[11323] := 16#9145;
   // UNICODE_TO_GBK[11324] := 16#6151;
   // UNICODE_TO_GBK[11325] := 16#C9E5;
   // UNICODE_TO_GBK[11326] := 16#6152;
   // UNICODE_TO_GBK[11327] := 16#9146;
   // UNICODE_TO_GBK[11328] := 16#6153;
   // UNICODE_TO_GBK[11329] := 16#9147;
   // UNICODE_TO_GBK[11330] := 16#6154;
   // UNICODE_TO_GBK[11331] := 16#9148;
   // UNICODE_TO_GBK[11332] := 16#6155;
   // UNICODE_TO_GBK[11333] := 16#C4BD;
   // UNICODE_TO_GBK[11334] := 16#6156;
   // UNICODE_TO_GBK[11335] := 16#9149;
   // UNICODE_TO_GBK[11336] := 16#6157;
   // UNICODE_TO_GBK[11337] := 16#914A;
   // UNICODE_TO_GBK[11338] := 16#6158;
   // UNICODE_TO_GBK[11339] := 16#914B;
   // UNICODE_TO_GBK[11340] := 16#6159;
   // UNICODE_TO_GBK[11341] := 16#914C;
   // UNICODE_TO_GBK[11342] := 16#615A;
   // UNICODE_TO_GBK[11343] := 16#914D;
   // UNICODE_TO_GBK[11344] := 16#615B;
   // UNICODE_TO_GBK[11345] := 16#914E;
   // UNICODE_TO_GBK[11346] := 16#615C;
   // UNICODE_TO_GBK[11347] := 16#914F;
   // UNICODE_TO_GBK[11348] := 16#615D;
   // UNICODE_TO_GBK[11349] := 16#EDAB;
   // UNICODE_TO_GBK[11350] := 16#615E;
   // UNICODE_TO_GBK[11351] := 16#9150;
   // UNICODE_TO_GBK[11352] := 16#615F;
   // UNICODE_TO_GBK[11353] := 16#9151;
   // UNICODE_TO_GBK[11354] := 16#6160;
   // UNICODE_TO_GBK[11355] := 16#9152;
   // UNICODE_TO_GBK[11356] := 16#6161;
   // UNICODE_TO_GBK[11357] := 16#9153;
   // UNICODE_TO_GBK[11358] := 16#6162;
   // UNICODE_TO_GBK[11359] := 16#C2FD;
   // UNICODE_TO_GBK[11360] := 16#6163;
   // UNICODE_TO_GBK[11361] := 16#9154;
   // UNICODE_TO_GBK[11362] := 16#6164;
   // UNICODE_TO_GBK[11363] := 16#9155;
   // UNICODE_TO_GBK[11364] := 16#6165;
   // UNICODE_TO_GBK[11365] := 16#9156;
   // UNICODE_TO_GBK[11366] := 16#6166;
   // UNICODE_TO_GBK[11367] := 16#9157;
   // UNICODE_TO_GBK[11368] := 16#6167;
   // UNICODE_TO_GBK[11369] := 16#BBDB;
   // UNICODE_TO_GBK[11370] := 16#6168;
   // UNICODE_TO_GBK[11371] := 16#BFAE;
   // UNICODE_TO_GBK[11372] := 16#6169;
   // UNICODE_TO_GBK[11373] := 16#9158;
   // UNICODE_TO_GBK[11374] := 16#616A;
   // UNICODE_TO_GBK[11375] := 16#9159;
   // UNICODE_TO_GBK[11376] := 16#616B;
   // UNICODE_TO_GBK[11377] := 16#915A;
   // UNICODE_TO_GBK[11378] := 16#616C;
   // UNICODE_TO_GBK[11379] := 16#915B;
   // UNICODE_TO_GBK[11380] := 16#616D;
   // UNICODE_TO_GBK[11381] := 16#915C;
   // UNICODE_TO_GBK[11382] := 16#616E;
   // UNICODE_TO_GBK[11383] := 16#915D;
   // UNICODE_TO_GBK[11384] := 16#616F;
   // UNICODE_TO_GBK[11385] := 16#915E;
   // UNICODE_TO_GBK[11386] := 16#6170;
   // UNICODE_TO_GBK[11387] := 16#CEBF;
   // UNICODE_TO_GBK[11388] := 16#6171;
   // UNICODE_TO_GBK[11389] := 16#915F;
   // UNICODE_TO_GBK[11390] := 16#6172;
   // UNICODE_TO_GBK[11391] := 16#9160;
   // UNICODE_TO_GBK[11392] := 16#6173;
   // UNICODE_TO_GBK[11393] := 16#9161;
   // UNICODE_TO_GBK[11394] := 16#6174;
   // UNICODE_TO_GBK[11395] := 16#9162;
   // UNICODE_TO_GBK[11396] := 16#6175;
   // UNICODE_TO_GBK[11397] := 16#E3BC;
   // UNICODE_TO_GBK[11398] := 16#6176;
   // UNICODE_TO_GBK[11399] := 16#9163;
   // UNICODE_TO_GBK[11400] := 16#6177;
   // UNICODE_TO_GBK[11401] := 16#BFB6;
   // UNICODE_TO_GBK[11402] := 16#6178;
   // UNICODE_TO_GBK[11403] := 16#9164;
   // UNICODE_TO_GBK[11404] := 16#6179;
   // UNICODE_TO_GBK[11405] := 16#9165;
   // UNICODE_TO_GBK[11406] := 16#617A;
   // UNICODE_TO_GBK[11407] := 16#9166;
   // UNICODE_TO_GBK[11408] := 16#617B;
   // UNICODE_TO_GBK[11409] := 16#9167;
   // UNICODE_TO_GBK[11410] := 16#617C;
   // UNICODE_TO_GBK[11411] := 16#9168;
   // UNICODE_TO_GBK[11412] := 16#617D;
   // UNICODE_TO_GBK[11413] := 16#9169;
   // UNICODE_TO_GBK[11414] := 16#617E;
   // UNICODE_TO_GBK[11415] := 16#916A;
   // UNICODE_TO_GBK[11416] := 16#617F;
   // UNICODE_TO_GBK[11417] := 16#916B;
   // UNICODE_TO_GBK[11418] := 16#6180;
   // UNICODE_TO_GBK[11419] := 16#916C;
   // UNICODE_TO_GBK[11420] := 16#6181;
   // UNICODE_TO_GBK[11421] := 16#916D;
   // UNICODE_TO_GBK[11422] := 16#6182;
   // UNICODE_TO_GBK[11423] := 16#916E;
   // UNICODE_TO_GBK[11424] := 16#6183;
   // UNICODE_TO_GBK[11425] := 16#916F;
   // UNICODE_TO_GBK[11426] := 16#6184;
   // UNICODE_TO_GBK[11427] := 16#9170;
   // UNICODE_TO_GBK[11428] := 16#6185;
   // UNICODE_TO_GBK[11429] := 16#9171;
   // UNICODE_TO_GBK[11430] := 16#6186;
   // UNICODE_TO_GBK[11431] := 16#9172;
   // UNICODE_TO_GBK[11432] := 16#6187;
   // UNICODE_TO_GBK[11433] := 16#9173;
   // UNICODE_TO_GBK[11434] := 16#6188;
   // UNICODE_TO_GBK[11435] := 16#9174;
   // UNICODE_TO_GBK[11436] := 16#6189;
   // UNICODE_TO_GBK[11437] := 16#9175;
   // UNICODE_TO_GBK[11438] := 16#618A;
   // UNICODE_TO_GBK[11439] := 16#9176;
   // UNICODE_TO_GBK[11440] := 16#618B;
   // UNICODE_TO_GBK[11441] := 16#B1EF;
   // UNICODE_TO_GBK[11442] := 16#618C;
   // UNICODE_TO_GBK[11443] := 16#9177;
   // UNICODE_TO_GBK[11444] := 16#618D;
   // UNICODE_TO_GBK[11445] := 16#9178;
   // UNICODE_TO_GBK[11446] := 16#618E;
   // UNICODE_TO_GBK[11447] := 16#D4F7;
   // UNICODE_TO_GBK[11448] := 16#618F;
   // UNICODE_TO_GBK[11449] := 16#9179;
   // UNICODE_TO_GBK[11450] := 16#6190;
   // UNICODE_TO_GBK[11451] := 16#917A;
   // UNICODE_TO_GBK[11452] := 16#6191;
   // UNICODE_TO_GBK[11453] := 16#917B;
   // UNICODE_TO_GBK[11454] := 16#6192;
   // UNICODE_TO_GBK[11455] := 16#917C;
   // UNICODE_TO_GBK[11456] := 16#6193;
   // UNICODE_TO_GBK[11457] := 16#917D;
   // UNICODE_TO_GBK[11458] := 16#6194;
   // UNICODE_TO_GBK[11459] := 16#E3BE;
   // UNICODE_TO_GBK[11460] := 16#6195;
   // UNICODE_TO_GBK[11461] := 16#917E;
   // UNICODE_TO_GBK[11462] := 16#6196;
   // UNICODE_TO_GBK[11463] := 16#9180;
   // UNICODE_TO_GBK[11464] := 16#6197;
   // UNICODE_TO_GBK[11465] := 16#9181;
   // UNICODE_TO_GBK[11466] := 16#6198;
   // UNICODE_TO_GBK[11467] := 16#9182;
   // UNICODE_TO_GBK[11468] := 16#6199;
   // UNICODE_TO_GBK[11469] := 16#9183;
   // UNICODE_TO_GBK[11470] := 16#619A;
   // UNICODE_TO_GBK[11471] := 16#9184;
   // UNICODE_TO_GBK[11472] := 16#619B;
   // UNICODE_TO_GBK[11473] := 16#9185;
   // UNICODE_TO_GBK[11474] := 16#619C;
   // UNICODE_TO_GBK[11475] := 16#9186;
   // UNICODE_TO_GBK[11476] := 16#619D;
   // UNICODE_TO_GBK[11477] := 16#EDAD;
   // UNICODE_TO_GBK[11478] := 16#619E;
   // UNICODE_TO_GBK[11479] := 16#9187;
   // UNICODE_TO_GBK[11480] := 16#619F;
   // UNICODE_TO_GBK[11481] := 16#9188;
   // UNICODE_TO_GBK[11482] := 16#61A0;
   // UNICODE_TO_GBK[11483] := 16#9189;
   // UNICODE_TO_GBK[11484] := 16#61A1;
   // UNICODE_TO_GBK[11485] := 16#918A;
   // UNICODE_TO_GBK[11486] := 16#61A2;
   // UNICODE_TO_GBK[11487] := 16#918B;
   // UNICODE_TO_GBK[11488] := 16#61A3;
   // UNICODE_TO_GBK[11489] := 16#918C;
   // UNICODE_TO_GBK[11490] := 16#61A4;
   // UNICODE_TO_GBK[11491] := 16#918D;
   // UNICODE_TO_GBK[11492] := 16#61A5;
   // UNICODE_TO_GBK[11493] := 16#918E;
   // UNICODE_TO_GBK[11494] := 16#61A6;
   // UNICODE_TO_GBK[11495] := 16#918F;
   // UNICODE_TO_GBK[11496] := 16#61A7;
   // UNICODE_TO_GBK[11497] := 16#E3BF;
   // UNICODE_TO_GBK[11498] := 16#61A8;
   // UNICODE_TO_GBK[11499] := 16#BAA9;
   // UNICODE_TO_GBK[11500] := 16#61A9;
   // UNICODE_TO_GBK[11501] := 16#EDAC;
   // UNICODE_TO_GBK[11502] := 16#61AA;
   // UNICODE_TO_GBK[11503] := 16#9190;
   // UNICODE_TO_GBK[11504] := 16#61AB;
   // UNICODE_TO_GBK[11505] := 16#9191;
   // UNICODE_TO_GBK[11506] := 16#61AC;
   // UNICODE_TO_GBK[11507] := 16#E3BD;
   // UNICODE_TO_GBK[11508] := 16#61AD;
   // UNICODE_TO_GBK[11509] := 16#9192;
   // UNICODE_TO_GBK[11510] := 16#61AE;
   // UNICODE_TO_GBK[11511] := 16#9193;
   // UNICODE_TO_GBK[11512] := 16#61AF;
   // UNICODE_TO_GBK[11513] := 16#9194;
   // UNICODE_TO_GBK[11514] := 16#61B0;
   // UNICODE_TO_GBK[11515] := 16#9195;
   // UNICODE_TO_GBK[11516] := 16#61B1;
   // UNICODE_TO_GBK[11517] := 16#9196;
   // UNICODE_TO_GBK[11518] := 16#61B2;
   // UNICODE_TO_GBK[11519] := 16#9197;
   // UNICODE_TO_GBK[11520] := 16#61B3;
   // UNICODE_TO_GBK[11521] := 16#9198;
   // UNICODE_TO_GBK[11522] := 16#61B4;
   // UNICODE_TO_GBK[11523] := 16#9199;
   // UNICODE_TO_GBK[11524] := 16#61B5;
   // UNICODE_TO_GBK[11525] := 16#919A;
   // UNICODE_TO_GBK[11526] := 16#61B6;
   // UNICODE_TO_GBK[11527] := 16#919B;
   // UNICODE_TO_GBK[11528] := 16#61B7;
   // UNICODE_TO_GBK[11529] := 16#E3C0;
   // UNICODE_TO_GBK[11530] := 16#61B8;
   // UNICODE_TO_GBK[11531] := 16#919C;
   // UNICODE_TO_GBK[11532] := 16#61B9;
   // UNICODE_TO_GBK[11533] := 16#919D;
   // UNICODE_TO_GBK[11534] := 16#61BA;
   // UNICODE_TO_GBK[11535] := 16#919E;
   // UNICODE_TO_GBK[11536] := 16#61BB;
   // UNICODE_TO_GBK[11537] := 16#919F;
   // UNICODE_TO_GBK[11538] := 16#61BC;
   // UNICODE_TO_GBK[11539] := 16#91A0;
   // UNICODE_TO_GBK[11540] := 16#61BD;
   // UNICODE_TO_GBK[11541] := 16#91A1;
   // UNICODE_TO_GBK[11542] := 16#61BE;
   // UNICODE_TO_GBK[11543] := 16#BAB6;
   // UNICODE_TO_GBK[11544] := 16#61BF;
   // UNICODE_TO_GBK[11545] := 16#91A2;
   // UNICODE_TO_GBK[11546] := 16#61C0;
   // UNICODE_TO_GBK[11547] := 16#91A3;
   // UNICODE_TO_GBK[11548] := 16#61C1;
   // UNICODE_TO_GBK[11549] := 16#91A4;
   // UNICODE_TO_GBK[11550] := 16#61C2;
   // UNICODE_TO_GBK[11551] := 16#B6AE;
   // UNICODE_TO_GBK[11552] := 16#61C3;
   // UNICODE_TO_GBK[11553] := 16#91A5;
   // UNICODE_TO_GBK[11554] := 16#61C4;
   // UNICODE_TO_GBK[11555] := 16#91A6;
   // UNICODE_TO_GBK[11556] := 16#61C5;
   // UNICODE_TO_GBK[11557] := 16#91A7;
   // UNICODE_TO_GBK[11558] := 16#61C6;
   // UNICODE_TO_GBK[11559] := 16#91A8;
   // UNICODE_TO_GBK[11560] := 16#61C7;
   // UNICODE_TO_GBK[11561] := 16#91A9;
   // UNICODE_TO_GBK[11562] := 16#61C8;
   // UNICODE_TO_GBK[11563] := 16#D0B8;
   // UNICODE_TO_GBK[11564] := 16#61C9;
   // UNICODE_TO_GBK[11565] := 16#91AA;
   // UNICODE_TO_GBK[11566] := 16#61CA;
   // UNICODE_TO_GBK[11567] := 16#B0C3;
   // UNICODE_TO_GBK[11568] := 16#61CB;
   // UNICODE_TO_GBK[11569] := 16#EDAE;
   // UNICODE_TO_GBK[11570] := 16#61CC;
   // UNICODE_TO_GBK[11571] := 16#91AB;
   // UNICODE_TO_GBK[11572] := 16#61CD;
   // UNICODE_TO_GBK[11573] := 16#91AC;
   // UNICODE_TO_GBK[11574] := 16#61CE;
   // UNICODE_TO_GBK[11575] := 16#91AD;
   // UNICODE_TO_GBK[11576] := 16#61CF;
   // UNICODE_TO_GBK[11577] := 16#91AE;
   // UNICODE_TO_GBK[11578] := 16#61D0;
   // UNICODE_TO_GBK[11579] := 16#91AF;
   // UNICODE_TO_GBK[11580] := 16#61D1;
   // UNICODE_TO_GBK[11581] := 16#EDAF;
   // UNICODE_TO_GBK[11582] := 16#61D2;
   // UNICODE_TO_GBK[11583] := 16#C0C1;
   // UNICODE_TO_GBK[11584] := 16#61D3;
   // UNICODE_TO_GBK[11585] := 16#91B0;
   // UNICODE_TO_GBK[11586] := 16#61D4;
   // UNICODE_TO_GBK[11587] := 16#E3C1;
   // UNICODE_TO_GBK[11588] := 16#61D5;
   // UNICODE_TO_GBK[11589] := 16#91B1;
   // UNICODE_TO_GBK[11590] := 16#61D6;
   // UNICODE_TO_GBK[11591] := 16#91B2;
   // UNICODE_TO_GBK[11592] := 16#61D7;
   // UNICODE_TO_GBK[11593] := 16#91B3;
   // UNICODE_TO_GBK[11594] := 16#61D8;
   // UNICODE_TO_GBK[11595] := 16#91B4;
   // UNICODE_TO_GBK[11596] := 16#61D9;
   // UNICODE_TO_GBK[11597] := 16#91B5;
   // UNICODE_TO_GBK[11598] := 16#61DA;
   // UNICODE_TO_GBK[11599] := 16#91B6;
   // UNICODE_TO_GBK[11600] := 16#61DB;
   // UNICODE_TO_GBK[11601] := 16#91B7;
   // UNICODE_TO_GBK[11602] := 16#61DC;
   // UNICODE_TO_GBK[11603] := 16#91B8;
   // UNICODE_TO_GBK[11604] := 16#61DD;
   // UNICODE_TO_GBK[11605] := 16#91B9;
   // UNICODE_TO_GBK[11606] := 16#61DE;
   // UNICODE_TO_GBK[11607] := 16#91BA;
   // UNICODE_TO_GBK[11608] := 16#61DF;
   // UNICODE_TO_GBK[11609] := 16#91BB;
   // UNICODE_TO_GBK[11610] := 16#61E0;
   // UNICODE_TO_GBK[11611] := 16#91BC;
   // UNICODE_TO_GBK[11612] := 16#61E1;
   // UNICODE_TO_GBK[11613] := 16#91BD;
   // UNICODE_TO_GBK[11614] := 16#61E2;
   // UNICODE_TO_GBK[11615] := 16#91BE;
   // UNICODE_TO_GBK[11616] := 16#61E3;
   // UNICODE_TO_GBK[11617] := 16#91BF;
   // UNICODE_TO_GBK[11618] := 16#61E4;
   // UNICODE_TO_GBK[11619] := 16#91C0;
   // UNICODE_TO_GBK[11620] := 16#61E5;
   // UNICODE_TO_GBK[11621] := 16#91C1;
   // UNICODE_TO_GBK[11622] := 16#61E6;
   // UNICODE_TO_GBK[11623] := 16#C5B3;
   // UNICODE_TO_GBK[11624] := 16#61E7;
   // UNICODE_TO_GBK[11625] := 16#91C2;
   // UNICODE_TO_GBK[11626] := 16#61E8;
   // UNICODE_TO_GBK[11627] := 16#91C3;
   // UNICODE_TO_GBK[11628] := 16#61E9;
   // UNICODE_TO_GBK[11629] := 16#91C4;
   // UNICODE_TO_GBK[11630] := 16#61EA;
   // UNICODE_TO_GBK[11631] := 16#91C5;
   // UNICODE_TO_GBK[11632] := 16#61EB;
   // UNICODE_TO_GBK[11633] := 16#91C6;
   // UNICODE_TO_GBK[11634] := 16#61EC;
   // UNICODE_TO_GBK[11635] := 16#91C7;
   // UNICODE_TO_GBK[11636] := 16#61ED;
   // UNICODE_TO_GBK[11637] := 16#91C8;
   // UNICODE_TO_GBK[11638] := 16#61EE;
   // UNICODE_TO_GBK[11639] := 16#91C9;
   // UNICODE_TO_GBK[11640] := 16#61EF;
   // UNICODE_TO_GBK[11641] := 16#91CA;
   // UNICODE_TO_GBK[11642] := 16#61F0;
   // UNICODE_TO_GBK[11643] := 16#91CB;
   // UNICODE_TO_GBK[11644] := 16#61F1;
   // UNICODE_TO_GBK[11645] := 16#91CC;
   // UNICODE_TO_GBK[11646] := 16#61F2;
   // UNICODE_TO_GBK[11647] := 16#91CD;
   // UNICODE_TO_GBK[11648] := 16#61F3;
   // UNICODE_TO_GBK[11649] := 16#91CE;
   // UNICODE_TO_GBK[11650] := 16#61F4;
   // UNICODE_TO_GBK[11651] := 16#91CF;
   // UNICODE_TO_GBK[11652] := 16#61F5;
   // UNICODE_TO_GBK[11653] := 16#E3C2;
   // UNICODE_TO_GBK[11654] := 16#61F6;
   // UNICODE_TO_GBK[11655] := 16#91D0;
   // UNICODE_TO_GBK[11656] := 16#61F7;
   // UNICODE_TO_GBK[11657] := 16#91D1;
   // UNICODE_TO_GBK[11658] := 16#61F8;
   // UNICODE_TO_GBK[11659] := 16#91D2;
   // UNICODE_TO_GBK[11660] := 16#61F9;
   // UNICODE_TO_GBK[11661] := 16#91D3;
   // UNICODE_TO_GBK[11662] := 16#61FA;
   // UNICODE_TO_GBK[11663] := 16#91D4;
   // UNICODE_TO_GBK[11664] := 16#61FB;
   // UNICODE_TO_GBK[11665] := 16#91D5;
   // UNICODE_TO_GBK[11666] := 16#61FC;
   // UNICODE_TO_GBK[11667] := 16#91D6;
   // UNICODE_TO_GBK[11668] := 16#61FD;
   // UNICODE_TO_GBK[11669] := 16#91D7;
   // UNICODE_TO_GBK[11670] := 16#61FE;
   // UNICODE_TO_GBK[11671] := 16#91D8;
   // UNICODE_TO_GBK[11672] := 16#61FF;
   // UNICODE_TO_GBK[11673] := 16#DCB2;
   // UNICODE_TO_GBK[11674] := 16#6200;
   // UNICODE_TO_GBK[11675] := 16#91D9;
   // UNICODE_TO_GBK[11676] := 16#6201;
   // UNICODE_TO_GBK[11677] := 16#91DA;
   // UNICODE_TO_GBK[11678] := 16#6202;
   // UNICODE_TO_GBK[11679] := 16#91DB;
   // UNICODE_TO_GBK[11680] := 16#6203;
   // UNICODE_TO_GBK[11681] := 16#91DC;
   // UNICODE_TO_GBK[11682] := 16#6204;
   // UNICODE_TO_GBK[11683] := 16#91DD;
   // UNICODE_TO_GBK[11684] := 16#6205;
   // UNICODE_TO_GBK[11685] := 16#91DE;
   // UNICODE_TO_GBK[11686] := 16#6206;
   // UNICODE_TO_GBK[11687] := 16#EDB0;
   // UNICODE_TO_GBK[11688] := 16#6207;
   // UNICODE_TO_GBK[11689] := 16#91DF;
   // UNICODE_TO_GBK[11690] := 16#6208;
   // UNICODE_TO_GBK[11691] := 16#B8EA;
   // UNICODE_TO_GBK[11692] := 16#6209;
   // UNICODE_TO_GBK[11693] := 16#91E0;
   // UNICODE_TO_GBK[11694] := 16#620A;
   // UNICODE_TO_GBK[11695] := 16#CEEC;
   // UNICODE_TO_GBK[11696] := 16#620B;
   // UNICODE_TO_GBK[11697] := 16#EAA7;
   // UNICODE_TO_GBK[11698] := 16#620C;
   // UNICODE_TO_GBK[11699] := 16#D0E7;
   // UNICODE_TO_GBK[11700] := 16#620D;
   // UNICODE_TO_GBK[11701] := 16#CAF9;
   // UNICODE_TO_GBK[11702] := 16#620E;
   // UNICODE_TO_GBK[11703] := 16#C8D6;
   // UNICODE_TO_GBK[11704] := 16#620F;
   // UNICODE_TO_GBK[11705] := 16#CFB7;
   // UNICODE_TO_GBK[11706] := 16#6210;
   // UNICODE_TO_GBK[11707] := 16#B3C9;
   // UNICODE_TO_GBK[11708] := 16#6211;
   // UNICODE_TO_GBK[11709] := 16#CED2;
   // UNICODE_TO_GBK[11710] := 16#6212;
   // UNICODE_TO_GBK[11711] := 16#BDE4;
   // UNICODE_TO_GBK[11712] := 16#6213;
   // UNICODE_TO_GBK[11713] := 16#91E1;
   // UNICODE_TO_GBK[11714] := 16#6214;
   // UNICODE_TO_GBK[11715] := 16#91E2;
   // UNICODE_TO_GBK[11716] := 16#6215;
   // UNICODE_TO_GBK[11717] := 16#E3DE;
   // UNICODE_TO_GBK[11718] := 16#6216;
   // UNICODE_TO_GBK[11719] := 16#BBF2;
   // UNICODE_TO_GBK[11720] := 16#6217;
   // UNICODE_TO_GBK[11721] := 16#EAA8;
   // UNICODE_TO_GBK[11722] := 16#6218;
   // UNICODE_TO_GBK[11723] := 16#D5BD;
   // UNICODE_TO_GBK[11724] := 16#6219;
   // UNICODE_TO_GBK[11725] := 16#91E3;
   // UNICODE_TO_GBK[11726] := 16#621A;
   // UNICODE_TO_GBK[11727] := 16#C6DD;
   // UNICODE_TO_GBK[11728] := 16#621B;
   // UNICODE_TO_GBK[11729] := 16#EAA9;
   // UNICODE_TO_GBK[11730] := 16#621C;
   // UNICODE_TO_GBK[11731] := 16#91E4;
   // UNICODE_TO_GBK[11732] := 16#621D;
   // UNICODE_TO_GBK[11733] := 16#91E5;
   // UNICODE_TO_GBK[11734] := 16#621E;
   // UNICODE_TO_GBK[11735] := 16#91E6;
   // UNICODE_TO_GBK[11736] := 16#621F;
   // UNICODE_TO_GBK[11737] := 16#EAAA;
   // UNICODE_TO_GBK[11738] := 16#6220;
   // UNICODE_TO_GBK[11739] := 16#91E7;
   // UNICODE_TO_GBK[11740] := 16#6221;
   // UNICODE_TO_GBK[11741] := 16#EAAC;
   // UNICODE_TO_GBK[11742] := 16#6222;
   // UNICODE_TO_GBK[11743] := 16#EAAB;
   // UNICODE_TO_GBK[11744] := 16#6223;
   // UNICODE_TO_GBK[11745] := 16#91E8;
   // UNICODE_TO_GBK[11746] := 16#6224;
   // UNICODE_TO_GBK[11747] := 16#EAAE;
   // UNICODE_TO_GBK[11748] := 16#6225;
   // UNICODE_TO_GBK[11749] := 16#EAAD;
   // UNICODE_TO_GBK[11750] := 16#6226;
   // UNICODE_TO_GBK[11751] := 16#91E9;
   // UNICODE_TO_GBK[11752] := 16#6227;
   // UNICODE_TO_GBK[11753] := 16#91EA;
   // UNICODE_TO_GBK[11754] := 16#6228;
   // UNICODE_TO_GBK[11755] := 16#91EB;
   // UNICODE_TO_GBK[11756] := 16#6229;
   // UNICODE_TO_GBK[11757] := 16#91EC;
   // UNICODE_TO_GBK[11758] := 16#622A;
   // UNICODE_TO_GBK[11759] := 16#BDD8;
   // UNICODE_TO_GBK[11760] := 16#622B;
   // UNICODE_TO_GBK[11761] := 16#91ED;
   // UNICODE_TO_GBK[11762] := 16#622C;
   // UNICODE_TO_GBK[11763] := 16#EAAF;
   // UNICODE_TO_GBK[11764] := 16#622D;
   // UNICODE_TO_GBK[11765] := 16#91EE;
   // UNICODE_TO_GBK[11766] := 16#622E;
   // UNICODE_TO_GBK[11767] := 16#C2BE;
   // UNICODE_TO_GBK[11768] := 16#622F;
   // UNICODE_TO_GBK[11769] := 16#91EF;
   // UNICODE_TO_GBK[11770] := 16#6230;
   // UNICODE_TO_GBK[11771] := 16#91F0;
   // UNICODE_TO_GBK[11772] := 16#6231;
   // UNICODE_TO_GBK[11773] := 16#91F1;
   // UNICODE_TO_GBK[11774] := 16#6232;
   // UNICODE_TO_GBK[11775] := 16#91F2;
   // UNICODE_TO_GBK[11776] := 16#6233;
   // UNICODE_TO_GBK[11777] := 16#B4C1;
   // UNICODE_TO_GBK[11778] := 16#6234;
   // UNICODE_TO_GBK[11779] := 16#B4F7;
   // UNICODE_TO_GBK[11780] := 16#6235;
   // UNICODE_TO_GBK[11781] := 16#91F3;
   // UNICODE_TO_GBK[11782] := 16#6236;
   // UNICODE_TO_GBK[11783] := 16#91F4;
   // UNICODE_TO_GBK[11784] := 16#6237;
   // UNICODE_TO_GBK[11785] := 16#BBA7;
   // UNICODE_TO_GBK[11786] := 16#6238;
   // UNICODE_TO_GBK[11787] := 16#91F5;
   // UNICODE_TO_GBK[11788] := 16#6239;
   // UNICODE_TO_GBK[11789] := 16#91F6;
   // UNICODE_TO_GBK[11790] := 16#623A;
   // UNICODE_TO_GBK[11791] := 16#91F7;
   // UNICODE_TO_GBK[11792] := 16#623B;
   // UNICODE_TO_GBK[11793] := 16#91F8;
   // UNICODE_TO_GBK[11794] := 16#623C;
   // UNICODE_TO_GBK[11795] := 16#91F9;
   // UNICODE_TO_GBK[11796] := 16#623D;
   // UNICODE_TO_GBK[11797] := 16#ECE6;
   // UNICODE_TO_GBK[11798] := 16#623E;
   // UNICODE_TO_GBK[11799] := 16#ECE5;
   // UNICODE_TO_GBK[11800] := 16#623F;
   // UNICODE_TO_GBK[11801] := 16#B7BF;
   // UNICODE_TO_GBK[11802] := 16#6240;
   // UNICODE_TO_GBK[11803] := 16#CBF9;
   // UNICODE_TO_GBK[11804] := 16#6241;
   // UNICODE_TO_GBK[11805] := 16#B1E2;
   // UNICODE_TO_GBK[11806] := 16#6242;
   // UNICODE_TO_GBK[11807] := 16#91FA;
   // UNICODE_TO_GBK[11808] := 16#6243;
   // UNICODE_TO_GBK[11809] := 16#ECE7;
   // UNICODE_TO_GBK[11810] := 16#6244;
   // UNICODE_TO_GBK[11811] := 16#91FB;
   // UNICODE_TO_GBK[11812] := 16#6245;
   // UNICODE_TO_GBK[11813] := 16#91FC;
   // UNICODE_TO_GBK[11814] := 16#6246;
   // UNICODE_TO_GBK[11815] := 16#91FD;
   // UNICODE_TO_GBK[11816] := 16#6247;
   // UNICODE_TO_GBK[11817] := 16#C9C8;
   // UNICODE_TO_GBK[11818] := 16#6248;
   // UNICODE_TO_GBK[11819] := 16#ECE8;
   // UNICODE_TO_GBK[11820] := 16#6249;
   // UNICODE_TO_GBK[11821] := 16#ECE9;
   // UNICODE_TO_GBK[11822] := 16#624A;
   // UNICODE_TO_GBK[11823] := 16#91FE;
   // UNICODE_TO_GBK[11824] := 16#624B;
   // UNICODE_TO_GBK[11825] := 16#CAD6;
   // UNICODE_TO_GBK[11826] := 16#624C;
   // UNICODE_TO_GBK[11827] := 16#DED0;
   // UNICODE_TO_GBK[11828] := 16#624D;
   // UNICODE_TO_GBK[11829] := 16#B2C5;
   // UNICODE_TO_GBK[11830] := 16#624E;
   // UNICODE_TO_GBK[11831] := 16#D4FA;
   // UNICODE_TO_GBK[11832] := 16#624F;
   // UNICODE_TO_GBK[11833] := 16#9240;
   // UNICODE_TO_GBK[11834] := 16#6250;
   // UNICODE_TO_GBK[11835] := 16#9241;
   // UNICODE_TO_GBK[11836] := 16#6251;
   // UNICODE_TO_GBK[11837] := 16#C6CB;
   // UNICODE_TO_GBK[11838] := 16#6252;
   // UNICODE_TO_GBK[11839] := 16#B0C7;
   // UNICODE_TO_GBK[11840] := 16#6253;
   // UNICODE_TO_GBK[11841] := 16#B4F2;
   // UNICODE_TO_GBK[11842] := 16#6254;
   // UNICODE_TO_GBK[11843] := 16#C8D3;
   // UNICODE_TO_GBK[11844] := 16#6255;
   // UNICODE_TO_GBK[11845] := 16#9242;
   // UNICODE_TO_GBK[11846] := 16#6256;
   // UNICODE_TO_GBK[11847] := 16#9243;
   // UNICODE_TO_GBK[11848] := 16#6257;
   // UNICODE_TO_GBK[11849] := 16#9244;
   // UNICODE_TO_GBK[11850] := 16#6258;
   // UNICODE_TO_GBK[11851] := 16#CDD0;
   // UNICODE_TO_GBK[11852] := 16#6259;
   // UNICODE_TO_GBK[11853] := 16#9245;
   // UNICODE_TO_GBK[11854] := 16#625A;
   // UNICODE_TO_GBK[11855] := 16#9246;
   // UNICODE_TO_GBK[11856] := 16#625B;
   // UNICODE_TO_GBK[11857] := 16#BFB8;
   // UNICODE_TO_GBK[11858] := 16#625C;
   // UNICODE_TO_GBK[11859] := 16#9247;
   // UNICODE_TO_GBK[11860] := 16#625D;
   // UNICODE_TO_GBK[11861] := 16#9248;
   // UNICODE_TO_GBK[11862] := 16#625E;
   // UNICODE_TO_GBK[11863] := 16#9249;
   // UNICODE_TO_GBK[11864] := 16#625F;
   // UNICODE_TO_GBK[11865] := 16#924A;
   // UNICODE_TO_GBK[11866] := 16#6260;
   // UNICODE_TO_GBK[11867] := 16#924B;
   // UNICODE_TO_GBK[11868] := 16#6261;
   // UNICODE_TO_GBK[11869] := 16#924C;
   // UNICODE_TO_GBK[11870] := 16#6262;
   // UNICODE_TO_GBK[11871] := 16#924D;
   // UNICODE_TO_GBK[11872] := 16#6263;
   // UNICODE_TO_GBK[11873] := 16#BFDB;
   // UNICODE_TO_GBK[11874] := 16#6264;
   // UNICODE_TO_GBK[11875] := 16#924E;
   // UNICODE_TO_GBK[11876] := 16#6265;
   // UNICODE_TO_GBK[11877] := 16#924F;
   // UNICODE_TO_GBK[11878] := 16#6266;
   // UNICODE_TO_GBK[11879] := 16#C7A4;
   // UNICODE_TO_GBK[11880] := 16#6267;
   // UNICODE_TO_GBK[11881] := 16#D6B4;
   // UNICODE_TO_GBK[11882] := 16#6268;
   // UNICODE_TO_GBK[11883] := 16#9250;
   // UNICODE_TO_GBK[11884] := 16#6269;
   // UNICODE_TO_GBK[11885] := 16#C0A9;
   // UNICODE_TO_GBK[11886] := 16#626A;
   // UNICODE_TO_GBK[11887] := 16#DED1;
   // UNICODE_TO_GBK[11888] := 16#626B;
   // UNICODE_TO_GBK[11889] := 16#C9A8;
   // UNICODE_TO_GBK[11890] := 16#626C;
   // UNICODE_TO_GBK[11891] := 16#D1EF;
   // UNICODE_TO_GBK[11892] := 16#626D;
   // UNICODE_TO_GBK[11893] := 16#C5A4;
   // UNICODE_TO_GBK[11894] := 16#626E;
   // UNICODE_TO_GBK[11895] := 16#B0E7;
   // UNICODE_TO_GBK[11896] := 16#626F;
   // UNICODE_TO_GBK[11897] := 16#B3B6;
   // UNICODE_TO_GBK[11898] := 16#6270;
   // UNICODE_TO_GBK[11899] := 16#C8C5;
   // UNICODE_TO_GBK[11900] := 16#6271;
   // UNICODE_TO_GBK[11901] := 16#9251;
   // UNICODE_TO_GBK[11902] := 16#6272;
   // UNICODE_TO_GBK[11903] := 16#9252;
   // UNICODE_TO_GBK[11904] := 16#6273;
   // UNICODE_TO_GBK[11905] := 16#B0E2;
   // UNICODE_TO_GBK[11906] := 16#6274;
   // UNICODE_TO_GBK[11907] := 16#9253;
   // UNICODE_TO_GBK[11908] := 16#6275;
   // UNICODE_TO_GBK[11909] := 16#9254;
   // UNICODE_TO_GBK[11910] := 16#6276;
   // UNICODE_TO_GBK[11911] := 16#B7F6;
   // UNICODE_TO_GBK[11912] := 16#6277;
   // UNICODE_TO_GBK[11913] := 16#9255;
   // UNICODE_TO_GBK[11914] := 16#6278;
   // UNICODE_TO_GBK[11915] := 16#9256;
   // UNICODE_TO_GBK[11916] := 16#6279;
   // UNICODE_TO_GBK[11917] := 16#C5FA;
   // UNICODE_TO_GBK[11918] := 16#627A;
   // UNICODE_TO_GBK[11919] := 16#9257;
   // UNICODE_TO_GBK[11920] := 16#627B;
   // UNICODE_TO_GBK[11921] := 16#9258;
   // UNICODE_TO_GBK[11922] := 16#627C;
   // UNICODE_TO_GBK[11923] := 16#B6F3;
   // UNICODE_TO_GBK[11924] := 16#627D;
   // UNICODE_TO_GBK[11925] := 16#9259;
   // UNICODE_TO_GBK[11926] := 16#627E;
   // UNICODE_TO_GBK[11927] := 16#D5D2;
   // UNICODE_TO_GBK[11928] := 16#627F;
   // UNICODE_TO_GBK[11929] := 16#B3D0;
   // UNICODE_TO_GBK[11930] := 16#6280;
   // UNICODE_TO_GBK[11931] := 16#BCBC;
   // UNICODE_TO_GBK[11932] := 16#6281;
   // UNICODE_TO_GBK[11933] := 16#925A;
   // UNICODE_TO_GBK[11934] := 16#6282;
   // UNICODE_TO_GBK[11935] := 16#925B;
   // UNICODE_TO_GBK[11936] := 16#6283;
   // UNICODE_TO_GBK[11937] := 16#925C;
   // UNICODE_TO_GBK[11938] := 16#6284;
   // UNICODE_TO_GBK[11939] := 16#B3AD;
   // UNICODE_TO_GBK[11940] := 16#6285;
   // UNICODE_TO_GBK[11941] := 16#925D;
   // UNICODE_TO_GBK[11942] := 16#6286;
   // UNICODE_TO_GBK[11943] := 16#925E;
   // UNICODE_TO_GBK[11944] := 16#6287;
   // UNICODE_TO_GBK[11945] := 16#925F;
   // UNICODE_TO_GBK[11946] := 16#6288;
   // UNICODE_TO_GBK[11947] := 16#9260;
   // UNICODE_TO_GBK[11948] := 16#6289;
   // UNICODE_TO_GBK[11949] := 16#BEF1;
   // UNICODE_TO_GBK[11950] := 16#628A;
   // UNICODE_TO_GBK[11951] := 16#B0D1;
   // UNICODE_TO_GBK[11952] := 16#628B;
   // UNICODE_TO_GBK[11953] := 16#9261;
   // UNICODE_TO_GBK[11954] := 16#628C;
   // UNICODE_TO_GBK[11955] := 16#9262;
   // UNICODE_TO_GBK[11956] := 16#628D;
   // UNICODE_TO_GBK[11957] := 16#9263;
   // UNICODE_TO_GBK[11958] := 16#628E;
   // UNICODE_TO_GBK[11959] := 16#9264;
   // UNICODE_TO_GBK[11960] := 16#628F;
   // UNICODE_TO_GBK[11961] := 16#9265;
   // UNICODE_TO_GBK[11962] := 16#6290;
   // UNICODE_TO_GBK[11963] := 16#9266;
   // UNICODE_TO_GBK[11964] := 16#6291;
   // UNICODE_TO_GBK[11965] := 16#D2D6;
   // UNICODE_TO_GBK[11966] := 16#6292;
   // UNICODE_TO_GBK[11967] := 16#CAE3;
   // UNICODE_TO_GBK[11968] := 16#6293;
   // UNICODE_TO_GBK[11969] := 16#D7A5;
   // UNICODE_TO_GBK[11970] := 16#6294;
   // UNICODE_TO_GBK[11971] := 16#9267;
   // UNICODE_TO_GBK[11972] := 16#6295;
   // UNICODE_TO_GBK[11973] := 16#CDB6;
   // UNICODE_TO_GBK[11974] := 16#6296;
   // UNICODE_TO_GBK[11975] := 16#B6B6;
   // UNICODE_TO_GBK[11976] := 16#6297;
   // UNICODE_TO_GBK[11977] := 16#BFB9;
   // UNICODE_TO_GBK[11978] := 16#6298;
   // UNICODE_TO_GBK[11979] := 16#D5DB;
   // UNICODE_TO_GBK[11980] := 16#6299;
   // UNICODE_TO_GBK[11981] := 16#9268;
   // UNICODE_TO_GBK[11982] := 16#629A;
   // UNICODE_TO_GBK[11983] := 16#B8A7;
   // UNICODE_TO_GBK[11984] := 16#629B;
   // UNICODE_TO_GBK[11985] := 16#C5D7;
   // UNICODE_TO_GBK[11986] := 16#629C;
   // UNICODE_TO_GBK[11987] := 16#9269;
   // UNICODE_TO_GBK[11988] := 16#629D;
   // UNICODE_TO_GBK[11989] := 16#926A;
   // UNICODE_TO_GBK[11990] := 16#629E;
   // UNICODE_TO_GBK[11991] := 16#926B;
   // UNICODE_TO_GBK[11992] := 16#629F;
   // UNICODE_TO_GBK[11993] := 16#DED2;
   // UNICODE_TO_GBK[11994] := 16#62A0;
   // UNICODE_TO_GBK[11995] := 16#BFD9;
   // UNICODE_TO_GBK[11996] := 16#62A1;
   // UNICODE_TO_GBK[11997] := 16#C2D5;
   // UNICODE_TO_GBK[11998] := 16#62A2;
   // UNICODE_TO_GBK[11999] := 16#C7C0;
   // UNICODE_TO_GBK[12000] := 16#62A3;
   // UNICODE_TO_GBK[12001] := 16#926C;
   // UNICODE_TO_GBK[12002] := 16#62A4;
   // UNICODE_TO_GBK[12003] := 16#BBA4;
   // UNICODE_TO_GBK[12004] := 16#62A5;
   // UNICODE_TO_GBK[12005] := 16#B1A8;
   // UNICODE_TO_GBK[12006] := 16#62A6;
   // UNICODE_TO_GBK[12007] := 16#926D;
   // UNICODE_TO_GBK[12008] := 16#62A7;
   // UNICODE_TO_GBK[12009] := 16#926E;
   // UNICODE_TO_GBK[12010] := 16#62A8;
   // UNICODE_TO_GBK[12011] := 16#C5EA;
   // UNICODE_TO_GBK[12012] := 16#62A9;
   // UNICODE_TO_GBK[12013] := 16#926F;
   // UNICODE_TO_GBK[12014] := 16#62AA;
   // UNICODE_TO_GBK[12015] := 16#9270;
   // UNICODE_TO_GBK[12016] := 16#62AB;
   // UNICODE_TO_GBK[12017] := 16#C5FB;
   // UNICODE_TO_GBK[12018] := 16#62AC;
   // UNICODE_TO_GBK[12019] := 16#CCA7;
   // UNICODE_TO_GBK[12020] := 16#62AD;
   // UNICODE_TO_GBK[12021] := 16#9271;
   // UNICODE_TO_GBK[12022] := 16#62AE;
   // UNICODE_TO_GBK[12023] := 16#9272;
   // UNICODE_TO_GBK[12024] := 16#62AF;
   // UNICODE_TO_GBK[12025] := 16#9273;
   // UNICODE_TO_GBK[12026] := 16#62B0;
   // UNICODE_TO_GBK[12027] := 16#9274;
   // UNICODE_TO_GBK[12028] := 16#62B1;
   // UNICODE_TO_GBK[12029] := 16#B1A7;
   // UNICODE_TO_GBK[12030] := 16#62B2;
   // UNICODE_TO_GBK[12031] := 16#9275;
   // UNICODE_TO_GBK[12032] := 16#62B3;
   // UNICODE_TO_GBK[12033] := 16#9276;
   // UNICODE_TO_GBK[12034] := 16#62B4;
   // UNICODE_TO_GBK[12035] := 16#9277;
   // UNICODE_TO_GBK[12036] := 16#62B5;
   // UNICODE_TO_GBK[12037] := 16#B5D6;
   // UNICODE_TO_GBK[12038] := 16#62B6;
   // UNICODE_TO_GBK[12039] := 16#9278;
   // UNICODE_TO_GBK[12040] := 16#62B7;
   // UNICODE_TO_GBK[12041] := 16#9279;
   // UNICODE_TO_GBK[12042] := 16#62B8;
   // UNICODE_TO_GBK[12043] := 16#927A;
   // UNICODE_TO_GBK[12044] := 16#62B9;
   // UNICODE_TO_GBK[12045] := 16#C4A8;
   // UNICODE_TO_GBK[12046] := 16#62BA;
   // UNICODE_TO_GBK[12047] := 16#927B;
   // UNICODE_TO_GBK[12048] := 16#62BB;
   // UNICODE_TO_GBK[12049] := 16#DED3;
   // UNICODE_TO_GBK[12050] := 16#62BC;
   // UNICODE_TO_GBK[12051] := 16#D1BA;
   // UNICODE_TO_GBK[12052] := 16#62BD;
   // UNICODE_TO_GBK[12053] := 16#B3E9;
   // UNICODE_TO_GBK[12054] := 16#62BE;
   // UNICODE_TO_GBK[12055] := 16#927C;
   // UNICODE_TO_GBK[12056] := 16#62BF;
   // UNICODE_TO_GBK[12057] := 16#C3F2;
   // UNICODE_TO_GBK[12058] := 16#62C0;
   // UNICODE_TO_GBK[12059] := 16#927D;
   // UNICODE_TO_GBK[12060] := 16#62C1;
   // UNICODE_TO_GBK[12061] := 16#927E;
   // UNICODE_TO_GBK[12062] := 16#62C2;
   // UNICODE_TO_GBK[12063] := 16#B7F7;
   // UNICODE_TO_GBK[12064] := 16#62C3;
   // UNICODE_TO_GBK[12065] := 16#9280;
   // UNICODE_TO_GBK[12066] := 16#62C4;
   // UNICODE_TO_GBK[12067] := 16#D6F4;
   // UNICODE_TO_GBK[12068] := 16#62C5;
   // UNICODE_TO_GBK[12069] := 16#B5A3;
   // UNICODE_TO_GBK[12070] := 16#62C6;
   // UNICODE_TO_GBK[12071] := 16#B2F0;
   // UNICODE_TO_GBK[12072] := 16#62C7;
   // UNICODE_TO_GBK[12073] := 16#C4B4;
   // UNICODE_TO_GBK[12074] := 16#62C8;
   // UNICODE_TO_GBK[12075] := 16#C4E9;
   // UNICODE_TO_GBK[12076] := 16#62C9;
   // UNICODE_TO_GBK[12077] := 16#C0AD;
   // UNICODE_TO_GBK[12078] := 16#62CA;
   // UNICODE_TO_GBK[12079] := 16#DED4;
   // UNICODE_TO_GBK[12080] := 16#62CB;
   // UNICODE_TO_GBK[12081] := 16#9281;
   // UNICODE_TO_GBK[12082] := 16#62CC;
   // UNICODE_TO_GBK[12083] := 16#B0E8;
   // UNICODE_TO_GBK[12084] := 16#62CD;
   // UNICODE_TO_GBK[12085] := 16#C5C4;
   // UNICODE_TO_GBK[12086] := 16#62CE;
   // UNICODE_TO_GBK[12087] := 16#C1E0;
   // UNICODE_TO_GBK[12088] := 16#62CF;
   // UNICODE_TO_GBK[12089] := 16#9282;
   // UNICODE_TO_GBK[12090] := 16#62D0;
   // UNICODE_TO_GBK[12091] := 16#B9D5;
   // UNICODE_TO_GBK[12092] := 16#62D1;
   // UNICODE_TO_GBK[12093] := 16#9283;
   // UNICODE_TO_GBK[12094] := 16#62D2;
   // UNICODE_TO_GBK[12095] := 16#BEDC;
   // UNICODE_TO_GBK[12096] := 16#62D3;
   // UNICODE_TO_GBK[12097] := 16#CDD8;
   // UNICODE_TO_GBK[12098] := 16#62D4;
   // UNICODE_TO_GBK[12099] := 16#B0CE;
   // UNICODE_TO_GBK[12100] := 16#62D5;
   // UNICODE_TO_GBK[12101] := 16#9284;
   // UNICODE_TO_GBK[12102] := 16#62D6;
   // UNICODE_TO_GBK[12103] := 16#CDCF;
   // UNICODE_TO_GBK[12104] := 16#62D7;
   // UNICODE_TO_GBK[12105] := 16#DED6;
   // UNICODE_TO_GBK[12106] := 16#62D8;
   // UNICODE_TO_GBK[12107] := 16#BED0;
   // UNICODE_TO_GBK[12108] := 16#62D9;
   // UNICODE_TO_GBK[12109] := 16#D7BE;
   // UNICODE_TO_GBK[12110] := 16#62DA;
   // UNICODE_TO_GBK[12111] := 16#DED5;
   // UNICODE_TO_GBK[12112] := 16#62DB;
   // UNICODE_TO_GBK[12113] := 16#D5D0;
   // UNICODE_TO_GBK[12114] := 16#62DC;
   // UNICODE_TO_GBK[12115] := 16#B0DD;
   // UNICODE_TO_GBK[12116] := 16#62DD;
   // UNICODE_TO_GBK[12117] := 16#9285;
   // UNICODE_TO_GBK[12118] := 16#62DE;
   // UNICODE_TO_GBK[12119] := 16#9286;
   // UNICODE_TO_GBK[12120] := 16#62DF;
   // UNICODE_TO_GBK[12121] := 16#C4E2;
   // UNICODE_TO_GBK[12122] := 16#62E0;
   // UNICODE_TO_GBK[12123] := 16#9287;
   // UNICODE_TO_GBK[12124] := 16#62E1;
   // UNICODE_TO_GBK[12125] := 16#9288;
   // UNICODE_TO_GBK[12126] := 16#62E2;
   // UNICODE_TO_GBK[12127] := 16#C2A3;
   // UNICODE_TO_GBK[12128] := 16#62E3;
   // UNICODE_TO_GBK[12129] := 16#BCF0;
   // UNICODE_TO_GBK[12130] := 16#62E4;
   // UNICODE_TO_GBK[12131] := 16#9289;
   // UNICODE_TO_GBK[12132] := 16#62E5;
   // UNICODE_TO_GBK[12133] := 16#D3B5;
   // UNICODE_TO_GBK[12134] := 16#62E6;
   // UNICODE_TO_GBK[12135] := 16#C0B9;
   // UNICODE_TO_GBK[12136] := 16#62E7;
   // UNICODE_TO_GBK[12137] := 16#C5A1;
   // UNICODE_TO_GBK[12138] := 16#62E8;
   // UNICODE_TO_GBK[12139] := 16#B2A6;
   // UNICODE_TO_GBK[12140] := 16#62E9;
   // UNICODE_TO_GBK[12141] := 16#D4F1;
   // UNICODE_TO_GBK[12142] := 16#62EA;
   // UNICODE_TO_GBK[12143] := 16#928A;
   // UNICODE_TO_GBK[12144] := 16#62EB;
   // UNICODE_TO_GBK[12145] := 16#928B;
   // UNICODE_TO_GBK[12146] := 16#62EC;
   // UNICODE_TO_GBK[12147] := 16#C0A8;
   // UNICODE_TO_GBK[12148] := 16#62ED;
   // UNICODE_TO_GBK[12149] := 16#CAC3;
   // UNICODE_TO_GBK[12150] := 16#62EE;
   // UNICODE_TO_GBK[12151] := 16#DED7;
   // UNICODE_TO_GBK[12152] := 16#62EF;
   // UNICODE_TO_GBK[12153] := 16#D5FC;
   // UNICODE_TO_GBK[12154] := 16#62F0;
   // UNICODE_TO_GBK[12155] := 16#928C;
   // UNICODE_TO_GBK[12156] := 16#62F1;
   // UNICODE_TO_GBK[12157] := 16#B9B0;
   // UNICODE_TO_GBK[12158] := 16#62F2;
   // UNICODE_TO_GBK[12159] := 16#928D;
   // UNICODE_TO_GBK[12160] := 16#62F3;
   // UNICODE_TO_GBK[12161] := 16#C8AD;
   // UNICODE_TO_GBK[12162] := 16#62F4;
   // UNICODE_TO_GBK[12163] := 16#CBA9;
   // UNICODE_TO_GBK[12164] := 16#62F5;
   // UNICODE_TO_GBK[12165] := 16#928E;
   // UNICODE_TO_GBK[12166] := 16#62F6;
   // UNICODE_TO_GBK[12167] := 16#DED9;
   // UNICODE_TO_GBK[12168] := 16#62F7;
   // UNICODE_TO_GBK[12169] := 16#BFBD;
   // UNICODE_TO_GBK[12170] := 16#62F8;
   // UNICODE_TO_GBK[12171] := 16#928F;
   // UNICODE_TO_GBK[12172] := 16#62F9;
   // UNICODE_TO_GBK[12173] := 16#9290;
   // UNICODE_TO_GBK[12174] := 16#62FA;
   // UNICODE_TO_GBK[12175] := 16#9291;
   // UNICODE_TO_GBK[12176] := 16#62FB;
   // UNICODE_TO_GBK[12177] := 16#9292;
   // UNICODE_TO_GBK[12178] := 16#62FC;
   // UNICODE_TO_GBK[12179] := 16#C6B4;
   // UNICODE_TO_GBK[12180] := 16#62FD;
   // UNICODE_TO_GBK[12181] := 16#D7A7;
   // UNICODE_TO_GBK[12182] := 16#62FE;
   // UNICODE_TO_GBK[12183] := 16#CAB0;
   // UNICODE_TO_GBK[12184] := 16#62FF;
   // UNICODE_TO_GBK[12185] := 16#C4C3;
   // UNICODE_TO_GBK[12186] := 16#6300;
   // UNICODE_TO_GBK[12187] := 16#9293;
   // UNICODE_TO_GBK[12188] := 16#6301;
   // UNICODE_TO_GBK[12189] := 16#B3D6;
   // UNICODE_TO_GBK[12190] := 16#6302;
   // UNICODE_TO_GBK[12191] := 16#B9D2;
   // UNICODE_TO_GBK[12192] := 16#6303;
   // UNICODE_TO_GBK[12193] := 16#9294;
   // UNICODE_TO_GBK[12194] := 16#6304;
   // UNICODE_TO_GBK[12195] := 16#9295;
   // UNICODE_TO_GBK[12196] := 16#6305;
   // UNICODE_TO_GBK[12197] := 16#9296;
   // UNICODE_TO_GBK[12198] := 16#6306;
   // UNICODE_TO_GBK[12199] := 16#9297;
   // UNICODE_TO_GBK[12200] := 16#6307;
   // UNICODE_TO_GBK[12201] := 16#D6B8;
   // UNICODE_TO_GBK[12202] := 16#6308;
   // UNICODE_TO_GBK[12203] := 16#EAFC;
   // UNICODE_TO_GBK[12204] := 16#6309;
   // UNICODE_TO_GBK[12205] := 16#B0B4;
   // UNICODE_TO_GBK[12206] := 16#630A;
   // UNICODE_TO_GBK[12207] := 16#9298;
   // UNICODE_TO_GBK[12208] := 16#630B;
   // UNICODE_TO_GBK[12209] := 16#9299;
   // UNICODE_TO_GBK[12210] := 16#630C;
   // UNICODE_TO_GBK[12211] := 16#929A;
   // UNICODE_TO_GBK[12212] := 16#630D;
   // UNICODE_TO_GBK[12213] := 16#929B;
   // UNICODE_TO_GBK[12214] := 16#630E;
   // UNICODE_TO_GBK[12215] := 16#BFE6;
   // UNICODE_TO_GBK[12216] := 16#630F;
   // UNICODE_TO_GBK[12217] := 16#929C;
   // UNICODE_TO_GBK[12218] := 16#6310;
   // UNICODE_TO_GBK[12219] := 16#929D;
   // UNICODE_TO_GBK[12220] := 16#6311;
   // UNICODE_TO_GBK[12221] := 16#CCF4;
   // UNICODE_TO_GBK[12222] := 16#6312;
   // UNICODE_TO_GBK[12223] := 16#929E;
   // UNICODE_TO_GBK[12224] := 16#6313;
   // UNICODE_TO_GBK[12225] := 16#929F;
   // UNICODE_TO_GBK[12226] := 16#6314;
   // UNICODE_TO_GBK[12227] := 16#92A0;
   // UNICODE_TO_GBK[12228] := 16#6315;
   // UNICODE_TO_GBK[12229] := 16#92A1;
   // UNICODE_TO_GBK[12230] := 16#6316;
   // UNICODE_TO_GBK[12231] := 16#CDDA;
   // UNICODE_TO_GBK[12232] := 16#6317;
   // UNICODE_TO_GBK[12233] := 16#92A2;
   // UNICODE_TO_GBK[12234] := 16#6318;
   // UNICODE_TO_GBK[12235] := 16#92A3;
   // UNICODE_TO_GBK[12236] := 16#6319;
   // UNICODE_TO_GBK[12237] := 16#92A4;
   // UNICODE_TO_GBK[12238] := 16#631A;
   // UNICODE_TO_GBK[12239] := 16#D6BF;
   // UNICODE_TO_GBK[12240] := 16#631B;
   // UNICODE_TO_GBK[12241] := 16#C2CE;
   // UNICODE_TO_GBK[12242] := 16#631C;
   // UNICODE_TO_GBK[12243] := 16#92A5;
   // UNICODE_TO_GBK[12244] := 16#631D;
   // UNICODE_TO_GBK[12245] := 16#CECE;
   // UNICODE_TO_GBK[12246] := 16#631E;
   // UNICODE_TO_GBK[12247] := 16#CCA2;
   // UNICODE_TO_GBK[12248] := 16#631F;
   // UNICODE_TO_GBK[12249] := 16#D0AE;
   // UNICODE_TO_GBK[12250] := 16#6320;
   // UNICODE_TO_GBK[12251] := 16#C4D3;
   // UNICODE_TO_GBK[12252] := 16#6321;
   // UNICODE_TO_GBK[12253] := 16#B5B2;
   // UNICODE_TO_GBK[12254] := 16#6322;
   // UNICODE_TO_GBK[12255] := 16#DED8;
   // UNICODE_TO_GBK[12256] := 16#6323;
   // UNICODE_TO_GBK[12257] := 16#D5F5;
   // UNICODE_TO_GBK[12258] := 16#6324;
   // UNICODE_TO_GBK[12259] := 16#BCB7;
   // UNICODE_TO_GBK[12260] := 16#6325;
   // UNICODE_TO_GBK[12261] := 16#BBD3;
   // UNICODE_TO_GBK[12262] := 16#6326;
   // UNICODE_TO_GBK[12263] := 16#92A6;
   // UNICODE_TO_GBK[12264] := 16#6327;
   // UNICODE_TO_GBK[12265] := 16#92A7;
   // UNICODE_TO_GBK[12266] := 16#6328;
   // UNICODE_TO_GBK[12267] := 16#B0A4;
   // UNICODE_TO_GBK[12268] := 16#6329;
   // UNICODE_TO_GBK[12269] := 16#92A8;
   // UNICODE_TO_GBK[12270] := 16#632A;
   // UNICODE_TO_GBK[12271] := 16#C5B2;
   // UNICODE_TO_GBK[12272] := 16#632B;
   // UNICODE_TO_GBK[12273] := 16#B4EC;
   // UNICODE_TO_GBK[12274] := 16#632C;
   // UNICODE_TO_GBK[12275] := 16#92A9;
   // UNICODE_TO_GBK[12276] := 16#632D;
   // UNICODE_TO_GBK[12277] := 16#92AA;
   // UNICODE_TO_GBK[12278] := 16#632E;
   // UNICODE_TO_GBK[12279] := 16#92AB;
   // UNICODE_TO_GBK[12280] := 16#632F;
   // UNICODE_TO_GBK[12281] := 16#D5F1;
   // UNICODE_TO_GBK[12282] := 16#6330;
   // UNICODE_TO_GBK[12283] := 16#92AC;
   // UNICODE_TO_GBK[12284] := 16#6331;
   // UNICODE_TO_GBK[12285] := 16#92AD;
   // UNICODE_TO_GBK[12286] := 16#6332;
   // UNICODE_TO_GBK[12287] := 16#EAFD;
   // UNICODE_TO_GBK[12288] := 16#6333;
   // UNICODE_TO_GBK[12289] := 16#92AE;
   // UNICODE_TO_GBK[12290] := 16#6334;
   // UNICODE_TO_GBK[12291] := 16#92AF;
   // UNICODE_TO_GBK[12292] := 16#6335;
   // UNICODE_TO_GBK[12293] := 16#92B0;
   // UNICODE_TO_GBK[12294] := 16#6336;
   // UNICODE_TO_GBK[12295] := 16#92B1;
   // UNICODE_TO_GBK[12296] := 16#6337;
   // UNICODE_TO_GBK[12297] := 16#92B2;
   // UNICODE_TO_GBK[12298] := 16#6338;
   // UNICODE_TO_GBK[12299] := 16#92B3;
   // UNICODE_TO_GBK[12300] := 16#6339;
   // UNICODE_TO_GBK[12301] := 16#DEDA;
   // UNICODE_TO_GBK[12302] := 16#633A;
   // UNICODE_TO_GBK[12303] := 16#CDA6;
   // UNICODE_TO_GBK[12304] := 16#633B;
   // UNICODE_TO_GBK[12305] := 16#92B4;
   // UNICODE_TO_GBK[12306] := 16#633C;
   // UNICODE_TO_GBK[12307] := 16#92B5;
   // UNICODE_TO_GBK[12308] := 16#633D;
   // UNICODE_TO_GBK[12309] := 16#CDEC;
   // UNICODE_TO_GBK[12310] := 16#633E;
   // UNICODE_TO_GBK[12311] := 16#92B6;
   // UNICODE_TO_GBK[12312] := 16#633F;
   // UNICODE_TO_GBK[12313] := 16#92B7;
   // UNICODE_TO_GBK[12314] := 16#6340;
   // UNICODE_TO_GBK[12315] := 16#92B8;
   // UNICODE_TO_GBK[12316] := 16#6341;
   // UNICODE_TO_GBK[12317] := 16#92B9;
   // UNICODE_TO_GBK[12318] := 16#6342;
   // UNICODE_TO_GBK[12319] := 16#CEE6;
   // UNICODE_TO_GBK[12320] := 16#6343;
   // UNICODE_TO_GBK[12321] := 16#DEDC;
   // UNICODE_TO_GBK[12322] := 16#6344;
   // UNICODE_TO_GBK[12323] := 16#92BA;
   // UNICODE_TO_GBK[12324] := 16#6345;
   // UNICODE_TO_GBK[12325] := 16#CDB1;
